        IF VI_Zone_Configs[L_Adaptive_Zone_i].zone >= 1 AND VI_Zone_Configs[L_Adaptive_Zone_i].zone <= 4 THEN
            L_Adaptive_Weight := L_Adaptive_Weight * 1.2;
        ELSIF VI_Zone_Configs[L_Adaptive_Zone_i].zone >= 9 THEN
            L_Adaptive_Weight := L_Adaptive_Weight * 0.7;
        END_IF;

        IF L_Adaptive_Weight > 2.0 THEN
            L_Adaptive_Weight := 2.0;
        ELSIF L_Adaptive_Weight < 0.2 THEN
            L_Adaptive_Weight := 0.2;
        END_IF;

        IF L_Adaptive_Delta > VO_Adaptive_Max_Delta THEN
            VO_Adaptive_Max_Delta := L_Adaptive_Delta;
        END_IF;

        L_Adaptive_Weighted_Sum := L_Adaptive_Weighted_Sum + (L_Adaptive_Delta * L_Adaptive_Weight);
        L_Adaptive_Weight_Total := L_Adaptive_Weight_Total + L_Adaptive_Weight;
    END_IF;
END_FOR;

IF L_Adaptive_Weight_Total > 0.0 THEN
    VO_Adaptive_Effective_Delta := L_Adaptive_Weighted_Sum / L_Adaptive_Weight_Total;
END_IF;

IF VO_Adaptive_Effective_Delta > 1.5 THEN
    VO_Adaptive_Correction := 2.0;
ELSIF VO_Adaptive_Effective_Delta > 0.7 THEN
    VO_Adaptive_Correction := 1.0;
ELSIF VO_Adaptive_Effective_Delta < -1.5 THEN
    VO_Adaptive_Correction := -2.0;
ELSIF VO_Adaptive_Effective_Delta < -0.7 THEN
    VO_Adaptive_Correction := -1.0;
ELSE
    VO_Adaptive_Correction := 0.0;
END_IF;

IF VO_Adaptive_Max_Delta > 2.5 AND VO_Adaptive_Correction < 2.0 THEN
    VO_Adaptive_Correction := 2.0;
END_IF;

VO_Target_Supply_Temp := VO_Target_Supply_Temp + VO_Adaptive_Correction;

IF VO_Target_Supply_Temp < 20.0 THEN
    VO_Target_Supply_Temp := 20.0;
ELSIF VO_Target_Supply_Temp > 45.0 THEN
    VO_Target_Supply_Temp := 45.0;
END_IF;

// >>> BULK_SYNC_ANCHOR: FB_Heating_Adaptive_Target <<<
          
END_FUNCTION_BLOCK

FUNCTION_BLOCK FB_Heating_Circuit_Control
  VAR_INPUT
    VI_System_Time_MS : UDINT;
    VI_Current_Hour : UINT;
    VI_IsActivePLC : BOOL;
    VI_Config : ST_Heating_Config;
    VI_Tariff : ST_Tariff_Config;
    VI_Scenario_Adjust : REAL;
  END_VAR
  VAR_OUTPUT
    VO_Zone_Valves : ARRAY[1..GVL_CONSTANTS.C_MAX_HEATING_CIRCUITS] OF BOOL;
    VO_Heating_Sensor_Fault : BOOL;
  END_VAR
  VAR_IN_OUT
    VI_Zone_Configs : ARRAY[1..GVL_CONSTANTS.C_MAX_HEATING_CIRCUITS] OF ST_FloorHeating_Circuit_Config;
    VI_Floor_Temps : ARRAY[1..GVL_CONSTANTS.C_MAX_HEATING_CIRCUITS] OF REAL;
    VI_Room_Temps : ARRAY[1..16] OF REAL;
    VI_Rule_Actions : ARRAY[1..GVL_CONSTANTS.C_MAX_RULES] OF ST_Rule_Action;
  END_VAR
  VAR
    L_i : INT;
    L_j : INT;
    L_Climate_Zone_ID : INT;
    L_Zone_Config : ST_FloorHeating_Circuit_Config;
    L_Current_Temp : REAL;
    L_Sensor_Error : BOOL;
    L_Floor_Controllers : ARRAY[1..GVL_CONSTANTS.C_MAX_HEATING_CIRCUITS] OF FB_FloorHeating_Controller;
    L_Overheat_Timer : ARRAY[1..GVL_CONSTANTS.C_MAX_HEATING_CIRCUITS] OF FB_System_Timer;
    fbFloorTempValidator : ARRAY[1..GVL_CONSTANTS.C_MAX_HEATING_CIRCUITS] OF FB_Analog_Validator;
    fbRoomTempValidator : ARRAY[1..16] OF FB_Analog_Validator;
  END_VAR

            // ==============================================================================
// Heating circuit control helper
//
// Internal refactoring helper for FB_Heating_System_Manager.
// Owns per-circuit sensor validation, temperature source fallback,
// floor-heating controller call, overheat shutdown, and rule action projection.
// ==============================================================================



VO_Heating_Sensor_Fault := FALSE;

FOR L_i := 1 TO GVL_CONSTANTS.C_MAX_HEATING_CIRCUITS DO
    fbFloorTempValidator[L_i](
        VI_Value := VI_Floor_Temps[L_i],
        VI_Min_Valid := -40.0,
        VI_Max_Valid := 120.0,
        VI_Fallback_Mode := 0
    );

    L_Climate_Zone_ID := VI_Zone_Configs[L_i].zone;
    IF L_Climate_Zone_ID >= 1 AND L_Climate_Zone_ID <= 16 THEN
        fbRoomTempValidator[L_Climate_Zone_ID](
            VI_Value := VI_Room_Temps[L_Climate_Zone_ID],
            VI_Min_Valid := -40.0,
            VI_Max_Valid := 120.0,
            VI_Fallback_Mode := 0
        );
    END_IF;

    // Floor overheat protection
    L_Overheat_Timer[L_i](
        IN := fbFloorTempValidator[L_i].VO_Value > VI_Config.Overheat_Threshold,
        PT := T#60s,
        VI_System_Time_MS := VI_System_Time_MS
    );

    L_Current_Temp := 0.0;
    L_Sensor_Error := FALSE;

    IF VI_Zone_Configs[L_i].control_type = 1 OR VI_Zone_Configs[L_i].control_type = 2 THEN
        // Primary: room air temperature
        IF (L_Climate_Zone_ID >= 1) AND (L_Climate_Zone_ID <= 16) AND (NOT fbRoomTempValidator[L_Climate_Zone_ID].VO_Error) THEN
            L_Current_Temp := fbRoomTempValidator[L_Climate_Zone_ID].VO_Value;
        ELSIF NOT fbFloorTempValidator[L_i].VO_Error THEN
            L_Current_Temp := fbFloorTempValidator[L_i].VO_Value;
        ELSE
            L_Sensor_Error := TRUE;
        END_IF;
    ELSE
        // Primary: floor temperature
        IF NOT fbFloorTempValidator[L_i].VO_Error THEN
            L_Current_Temp := fbFloorTempValidator[L_i].VO_Value;
        ELSIF (L_Climate_Zone_ID >= 1) AND (L_Climate_Zone_ID <= 16) AND (NOT fbRoomTempValidator[L_Climate_Zone_ID].VO_Error) THEN
            L_Current_Temp := fbRoomTempValidator[L_Climate_Zone_ID].VO_Value;
        ELSE
            L_Sensor_Error := TRUE;
        END_IF;
    END_IF;

    IF L_Sensor_Error THEN
        VO_Heating_Sensor_Fault := TRUE;
        VO_Zone_Valves[L_i] := FALSE;
    ELSE
        L_Zone_Config := VI_Zone_Configs[L_i];
        L_Zone_Config.design_temp := L_Zone_Config.design_temp + VI_Scenario_Adjust;

        L_Floor_Controllers[L_i](
            VI_Current_Temp := L_Current_Temp,
            VI_Config := L_Zone_Config,
            VI_Tariff := VI_Tariff,
            VI_Current_Hour := VI_Current_Hour,
            VI_IsActivePLC := VI_IsActivePLC,
            VI_System_Time_MS := VI_System_Time_MS,
            VO_Valve_Bool => VO_Zone_Valves[L_i]
        );
    END_IF;

    IF L_Overheat_Timer[L_i].Q THEN
        VO_Zone_Valves[L_i] := FALSE;
    END_IF;

    FOR L_j := 1 TO GVL_CONSTANTS.C_MAX_RULES DO
        IF VI_Rule_Actions[L_j].Active AND VI_Rule_Actions[L_j].Target_ID = L_i THEN
            IF VI_Rule_Actions[L_j].Action_Type = E_Rule_Action_Type.ACTION_SET_FLOOR_HEATING THEN
                VO_Zone_Valves[L_i] := (VI_Rule_Actions[L_j].Value > 0.5);
            END_IF;
        END_IF;
    END_FOR;
END_FOR;

// >>> BULK_SYNC_ANCHOR: FB_Heating_Circuit_Control <<<
          
END_FUNCTION_BLOCK

FUNCTION_BLOCK FB_Rule_Engine
  VAR_INPUT
    VI_System_Time_MS : UDINT;
    VI_IsActivePLC : BOOL;
    VI_Security_Armed : BOOL;
    VI_Current_Time : TOD;
    VI_Day_Of_Week : INT;
  END_VAR
  VAR_OUTPUT
    VO_Preheat_Request : BOOL;
    VO_Actions : ARRAY[1..GVL_CONSTANTS.C_MAX_RULES] OF ST_Rule_Action;
  END_VAR
  VAR_IN_OUT
    VI_Rules : ARRAY[1..GVL_CONSTANTS.C_MAX_RULES] OF ST_User_Rule;
    VI_Indoor_Temps : ARRAY[1..16] OF REAL;
    VI_Floor_Temps : ARRAY[1..8] OF REAL;
    VI_Humidities : ARRAY[1..16] OF REAL;
    VI_CO2_Levels : ARRAY[1..16] OF REAL;
    VI_Motion_Sensors : ARRAY[1..16] OF BOOL;
    VI_Door_Sensors : ARRAY[1..GVL_CONSTANTS.C_MAX_DOOR_SENSORS] OF BOOL;
    VI_Window_Sensors : ARRAY[1..16] OF BOOL;
    VI_Water_Sensors : ARRAY[1..GVL_CONSTANTS.C_MAX_FLOOD_SENSORS] OF BOOL;
    VI_Smoke_Sensors : ARRAY[1..GVL_CONSTANTS.C_MAX_SMOKE_SENSORS] OF BOOL;
    VI_Methane_Sensors : ARRAY[1..GVL_CONSTANTS.C_MAX_METHANE_SENSORS] OF REAL;
    VI_CO_Sensors : ARRAY[1..GVL_CONSTANTS.C_MAX_CO_SENSORS] OF REAL;
  END_VAR
  VAR
    L_i : INT;
    L_Condition_Met : BOOL;
    L_Current_Value : REAL;
    L_Triggers : ARRAY[1..GVL_CONSTANTS.C_MAX_RULES] OF R_TRIG;
    L_Trigger_Count : ARRAY[1..GVL_CONSTANTS.C_MAX_RULES] OF UINT;
    L_Last_Reset_Time : UDINT;
    L_Elapsed_Time : UDINT;
  END_VAR

            IF NOT VI_IsActivePLC THEN RETURN; END_IF;

VO_Preheat_Request := FALSE;


// Сброс счетчиков срабатываний каждую минуту (защита от циклических зависимостей/дребезга)
L_Elapsed_Time := (SEL(VI_System_Time_MS >= L_Last_Reset_Time, VI_System_Time_MS - L_Last_Reset_Time, (4294967295 - L_Last_Reset_Time) + VI_System_Time_MS + 1));

IF L_Elapsed_Time >= GVL_CONSTANTS.C_MS_IN_MINUTE THEN
    L_Last_Reset_Time := VI_System_Time_MS;
    FOR L_i := 1 TO GVL_CONSTANTS.C_MAX_RULES DO
        L_Trigger_Count[L_i] := 0;
    END_FOR;
END_IF;

FOR L_i := 1 TO GVL_CONSTANTS.C_MAX_RULES DO

    VO_Actions[L_i].Active := FALSE;
    IF VI_Rules[L_i].Enabled THEN
        L_Condition_Met := FALSE;
        L_Current_Value := 0.0;
        
        // Определение значения для проверки
        IF VI_Rules[L_i].Condition_Target_ID > 0 THEN
            CASE VI_Rules[L_i].Condition_Type OF
                E_Rule_Condition_Type.COND_AIR_TEMP: IF VI_Rules[L_i].Condition_Target_ID <= 16 THEN L_Current_Value := VI_Indoor_Temps[VI_Rules[L_i].Condition_Target_ID]; END_IF;
                E_Rule_Condition_Type.COND_FLOOR_TEMP: IF VI_Rules[L_i].Condition_Target_ID <= 8 THEN L_Current_Value := VI_Floor_Temps[VI_Rules[L_i].Condition_Target_ID]; END_IF;
                E_Rule_Condition_Type.COND_HUMIDITY: IF VI_Rules[L_i].Condition_Target_ID <= 16 THEN L_Current_Value := VI_Humidities[VI_Rules[L_i].Condition_Target_ID]; END_IF;
                E_Rule_Condition_Type.COND_CO2: IF VI_Rules[L_i].Condition_Target_ID <= 16 THEN L_Current_Value := VI_CO2_Levels[VI_Rules[L_i].Condition_Target_ID]; END_IF;
                E_Rule_Condition_Type.COND_MOTION: IF VI_Rules[L_i].Condition_Target_ID <= 16 THEN L_Current_Value := SEL(VI_Motion_Sensors[VI_Rules[L_i].Condition_Target_ID], 0.0, 1.0); END_IF;
                E_Rule_Condition_Type.COND_DOOR_WINDOW: 
                    IF VI_Rules[L_i].Condition_Target_ID <= GVL_CONSTANTS.C_MAX_DOOR_SENSORS THEN
                        L_Current_Value := SEL(VI_Door_Sensors[VI_Rules[L_i].Condition_Target_ID] OR VI_Window_Sensors[VI_Rules[L_i].Condition_Target_ID], 0.0, 1.0);
                    ELSIF VI_Rules[L_i].Condition_Target_ID <= 16 THEN
                        L_Current_Value := SEL(VI_Window_Sensors[VI_Rules[L_i].Condition_Target_ID], 0.0, 1.0);
                    END_IF;
                E_Rule_Condition_Type.COND_FLOOD: IF VI_Rules[L_i].Condition_Target_ID <= GVL_CONSTANTS.C_MAX_FLOOD_SENSORS THEN L_Current_Value := SEL(VI_Water_Sensors[VI_Rules[L_i].Condition_Target_ID], 0.0, 1.0); END_IF;
                E_Rule_Condition_Type.COND_SMOKE: IF VI_Rules[L_i].Condition_Target_ID <= GVL_CONSTANTS.C_MAX_SMOKE_SENSORS THEN L_Current_Value := SEL(VI_Smoke_Sensors[VI_Rules[L_i].Condition_Target_ID], 0.0, 1.0); END_IF;
                E_Rule_Condition_Type.COND_METHANE: IF VI_Rules[L_i].Condition_Target_ID <= GVL_CONSTANTS.C_MAX_METHANE_SENSORS THEN L_Current_Value := VI_Methane_Sensors[VI_Rules[L_i].Condition_Target_ID]; END_IF;
                E_Rule_Condition_Type.COND_CO: IF VI_Rules[L_i].Condition_Target_ID <= GVL_CONSTANTS.C_MAX_CO_SENSORS THEN L_Current_Value := VI_CO_Sensors[VI_Rules[L_i].Condition_Target_ID]; END_IF;
                E_Rule_Condition_Type.COND_TIME_OF_DAY: L_Current_Value := TO_REAL(TOD_TO_UDINT(VI_Current_Time) / GVL_CONSTANTS.C_MS_IN_MINUTE); // Время в минутах
                E_Rule_Condition_Type.COND_DAY_OF_WEEK: L_Current_Value := TO_REAL(VI_Day_Of_Week);
            END_CASE;
        ELSE
            IF VI_Rules[L_i].Condition_Type = E_Rule_Condition_Type.COND_TIME_OF_DAY THEN
                L_Current_Value := TO_REAL(TOD_TO_UDINT(VI_Current_Time) / GVL_CONSTANTS.C_MS_IN_MINUTE); // Время в минутах
            ELSIF VI_Rules[L_i].Condition_Type = E_Rule_Condition_Type.COND_DAY_OF_WEEK THEN
                L_Current_Value := TO_REAL(VI_Day_Of_Week);
            END_IF;
        END_IF;
        
        // Проверка условия
        CASE VI_Rules[L_i].Condition_Op OF
            E_Rule_Comparison.COMP_GT: L_Condition_Met := (L_Current_Value > VI_Rules[L_i].Condition_Value);
            E_Rule_Comparison.COMP_LT: L_Condition_Met := (L_Current_Value < VI_Rules[L_i].Condition_Value);
            E_Rule_Comparison.COMP_EQ: L_Condition_Met := (ABS(L_Current_Value - VI_Rules[L_i].Condition_Value) < 0.1);
            E_Rule_Comparison.COMP_GE: L_Condition_Met := (L_Current_Value >= VI_Rules[L_i].Condition_Value);
            E_Rule_Comparison.COMP_LE: L_Condition_Met := (L_Current_Value <= VI_Rules[L_i].Condition_Value);
            E_Rule_Comparison.COMP_IN_RANGE: L_Condition_Met := (L_Current_Value >= VI_Rules[L_i].Condition_Value) AND (L_Current_Value <= VI_Rules[L_i].Condition_Value_Max);
            E_Rule_Comparison.COMP_TRUE: L_Condition_Met := (L_Current_Value > 0.5);
            E_Rule_Comparison.COMP_FALSE: L_Condition_Met := (L_Current_Value < 0.5);
        END_CASE;
        
        // Формирование действия
        L_Triggers[L_i](CLK := L_Condition_Met);
        
        IF L_Triggers[L_i].Q THEN
            L_Trigger_Count[L_i] := L_Trigger_Count[L_i] + 1;
            IF L_Trigger_Count[L_i] > 10 THEN
                // ТЗ 13.5: Блокировка правила при слишком частом срабатывании (циклическая зависимость)
                VO_Actions[L_i].Active := FALSE;
                VO_Actions[L_i].Triggered := FALSE;
                CONTINUE; // Пропускаем выполнение
            END_IF;
        END_IF;
        
        IF L_Condition_Met AND (L_Trigger_Count[L_i] <= 10) THEN
            VO_Actions[L_i].Active := TRUE;
            VO_Actions[L_i].Triggered := L_Triggers[L_i].Q;
            VO_Actions[L_i].Action_Type := VI_Rules[L_i].Action_Type;
            VO_Actions[L_i].Target_ID := VI_Rules[L_i].Action_Target_ID;
            VO_Actions[L_i].Value := VI_Rules[L_i].Action_Value;
        END_IF;
    END_IF;
END_FOR;
// >>> BULK_SYNC_ANCHOR: FB_Rule_Engine <<<
          
END_FUNCTION_BLOCK

FUNCTION_BLOCK FB_Trend_Analyzer
  VAR_INPUT
    VI_Count : INT;
  END_VAR
  VAR_OUTPUT
    VO_Average : REAL;
    VO_Max : REAL;
    VO_Min : REAL;
    VO_Trend_Up : BOOL;
    VO_Trend_Down : BOOL;
  END_VAR
  VAR_IN_OUT
    VI_Data : ARRAY[1..GVL_CONSTANTS.C_MAX_TREND_DATA_POINTS] OF REAL;
  END_VAR
  VAR
    L_i : INT;
    L_Sum : REAL;
  END_VAR

            IF VI_Count > 0 AND VI_Count <= GVL_CONSTANTS.C_MAX_TREND_DATA_POINTS THEN
    VO_Max := VI_Data[1];
    VO_Min := VI_Data[1];
    L_Sum := 0.0;
    
    FOR L_i := 1 TO VI_Count DO
        IF VI_Data[L_i] > VO_Max THEN VO_Max := VI_Data[L_i]; END_IF;
        IF VI_Data[L_i] < VO_Min THEN VO_Min := VI_Data[L_i]; END_IF;
        L_Sum := L_Sum + VI_Data[L_i];
    END_FOR;
    
    VO_Average := L_Sum / INT_TO_REAL(VI_Count);
    
    IF VI_Count >= 2 THEN
        VO_Trend_Up := (VI_Data[VI_Count] > VI_Data[1]);
        VO_Trend_Down := (VI_Data[VI_Count] < VI_Data[1]);
    END_IF;
END_IF;
          
END_FUNCTION_BLOCK

FUNCTION_BLOCK FB_BlackBox_Recorder
  VAR_INPUT
    VI_Current_Data : ST_BlackBox_Record;
    VI_Freeze : BOOL;
  END_VAR
  VAR_OUTPUT
    VO_Frozen : BOOL;
    VO_Records_Count : INT;
  END_VAR
  VAR
    L_Write_Index : INT := 0;
    L_Initialized : BOOL := FALSE;
  END_VAR

            IF NOT L_Initialized THEN
    L_Write_Index := GVL_Retain.G_BlackBox_LastIndex;
    IF L_Write_Index < 0 OR L_Write_Index >= GVL_CONSTANTS.C_MAX_BLACKBOX_RECORDS THEN
        L_Write_Index := 0;
        GVL_Retain.G_BlackBox_LastIndex := 0;
    END_IF;
    L_Initialized := TRUE;
END_IF;

IF VI_Freeze THEN
    GVL_Retain.G_BlackBox_Frozen := TRUE;
END_IF;

VO_Frozen := GVL_Retain.G_BlackBox_Frozen;

IF NOT GVL_Retain.G_BlackBox_Frozen THEN
    GVL_Retain.G_BlackBox_Buffer[L_Write_Index] := VI_Current_Data;
    GVL_Retain.G_BlackBox_LastIndex := L_Write_Index;
    
    L_Write_Index := L_Write_Index + 1;
    IF L_Write_Index >= GVL_CONSTANTS.C_MAX_BLACKBOX_RECORDS THEN
        L_Write_Index := 0;
    END_IF;
END_IF;

VO_Records_Count := GVL_CONSTANTS.C_MAX_BLACKBOX_RECORDS; // Размер кольцевого буфера
// >>> BULK_SYNC_ANCHOR: FB_BlackBox_Recorder <<<
          
END_FUNCTION_BLOCK

FUNCTION_BLOCK FB_System_Init
  VAR_IN_OUT
    VIO_Local_State : ST_System_State_Snapshot;
    VIO_Remote_State : ST_System_State_Snapshot;
  END_VAR
  VAR
    L_i : INT;
  END_VAR

            // ==============================================================================
// System init helper
//
// Internal helper for PRG_System.
// Owns first-boot initialization of RETAIN runtime state.
// ==============================================================================



IF NOT GVL_Retain.G_Initialized THEN
    FOR L_i := 0 TO GVL_CONSTANTS.C_MAX_PRESENCE_HISTORY - 1 DO
        GVL_Retain.G_Presence_History[L_i] := 0;
    END_FOR;

    GVL_Retain.G_History_Write_Idx := 1;
    GVL_Retain.G_History_Total_Events := 0;

    FOR L_i := 1 TO GVL_CONSTANTS.C_MAX_BOILERS DO
        GVL_Retain.G_Boiler_Accumulated_MS[L_i] := 0;
        GVL_Retain.G_Boiler_Work_Seconds[L_i] := 0;
    END_FOR;

    FOR L_i := 1 TO GVL_CONSTANTS.C_MAX_MANIFOLDS DO
        GVL_Retain.G_Valve_Test_Results[L_i] := FALSE;
    END_FOR;

    VIO_Local_State.Version := 0;
    VIO_Remote_State.Version := 0;

    GVL_Retain.G_Initialized := TRUE;
END_IF;

// >>> BULK_SYNC_ANCHOR: FB_System_Init <<<
          
END_FUNCTION_BLOCK

FUNCTION_BLOCK FB_Safety_Manager
  VAR_INPUT
    VI_Gas_Alarm : BOOL;
    VI_Leak_Alarm : BOOL;
    VI_Smoke_Alarm : BOOL;
    VI_Reset : BOOL;
  END_VAR
  VAR_OUTPUT
    VO_Gas_Latched : BOOL;
    VO_Leak_Latched : BOOL;
    VO_Smoke_Latched : BOOL;
    VO_Emergency_Stop : BOOL;
  END_VAR
  VAR
    L_Any_Active : BOOL;
  END_VAR

            // Защёлкиваем аварии независимо друг от друга
IF VI_Gas_Alarm THEN
    VO_Gas_Latched := TRUE;
END_IF;

IF VI_Leak_Alarm THEN
    VO_Leak_Latched := TRUE;
END_IF;

IF VI_Smoke_Alarm THEN
    VO_Smoke_Latched := TRUE;
END_IF;

L_Any_Active := VI_Gas_Alarm OR VI_Leak_Alarm OR VI_Smoke_Alarm;

// Ручной сброс допустим только когда все входные аварийные сигналы уже исчезли
IF VI_Reset AND NOT L_Any_Active THEN
    VO_Gas_Latched := FALSE;
    VO_Leak_Latched := FALSE;
    VO_Smoke_Latched := FALSE;
END_IF;

// Агрегированный аварийный стоп = любая защёлкнутая safety-авария
VO_Emergency_Stop := VO_Gas_Latched OR VO_Leak_Latched OR VO_Smoke_Latched;

// >>> BULK_SYNC_ANCHOR: FB_Safety_Manager <<<
          
END_FUNCTION_BLOCK

FUNCTION_BLOCK FB_System_Recovery
  VAR_IN_OUT
    VIO_Recovery_Done : BOOL;
  END_VAR

            // ==============================================================================
// System recovery helper
//
// Internal helper for PRG_System.
// Owns one-shot recovery of persistent safety/system state after boot.
// ==============================================================================



IF NOT VIO_Recovery_Done THEN
    IF GVL_PERSISTENT.P_Valid THEN
        GVL_STATE.G_Safety_Gas_Latched := GVL_PERSISTENT.P_Safety_Gas_Latched;
        GVL_STATE.G_Safety_Smoke_Latched := GVL_PERSISTENT.P_Safety_Smoke_Latched;
        GVL_STATE.G_Safety_Leak_Latched := GVL_PERSISTENT.P_Safety_Leak_Latched;
        GVL_STATE.G_System_Mode := GVL_PERSISTENT.P_System_Mode;
    END_IF;

    VIO_Recovery_Done := TRUE;
END_IF;

// >>> BULK_SYNC_ANCHOR: FB_System_Recovery <<<
          
END_FUNCTION_BLOCK

FUNCTION_BLOCK FB_System_Coordinator
  VAR_INPUT
    VI_Fire_Latched : BOOL;
    VI_Gas_Latched : BOOL;
    VI_Leak_Latched : BOOL;
    VI_IO_Degraded : BOOL;
    VI_Ownership_Violation : BOOL;
    VI_Behavior_Mode : E_Behavior_Mode;
  END_VAR
  VAR_OUTPUT
    VO_Block_Heating : BOOL;
    VO_Block_Ventilation : BOOL;
    VO_Block_Lighting : BOOL;
    VO_Block_Sockets : BOOL;
    VO_System_Degraded : BOOL;
    VO_Code : UDINT;
  END_VAR

            // reset
VO_Block_Heating := FALSE;
VO_Block_Ventilation := FALSE;
VO_Block_Lighting := FALSE;
VO_Block_Sockets := FALSE;
VO_System_Degraded := FALSE;
VO_Code := 0;

// FIRE has highest priority. Safety-stop ownership remains in PRG_Safety.
IF VI_Fire_Latched THEN
    VO_Block_Heating := TRUE;
    VO_Block_Ventilation := TRUE;
    VO_Block_Sockets := TRUE;
    VO_Code := 100;
    RETURN;
END_IF;

// GAS has higher priority than behavior mode.
IF VI_Gas_Latched THEN
    VO_Block_Heating := TRUE;
    VO_Block_Lighting := TRUE;
    VO_Block_Sockets := TRUE;
    VO_Code := 200;
    RETURN;
END_IF;

// LEAK blocks heating but does not suppress later degradation/mode overlays.
IF VI_Leak_Latched THEN
    VO_Block_Heating := TRUE;
    VO_Code := 300;
END_IF;

// IO degraded blocks heating and marks system degraded.
IF VI_IO_Degraded THEN
    VO_System_Degraded := TRUE;
    VO_Block_Heating := TRUE;
    IF VO_Code = 0 THEN
        VO_Code := 400;
    END_IF;
END_IF;

// Ownership violation marks system degraded. Test/result handler owns any safe-stop reaction.
IF VI_Ownership_Violation THEN
    VO_System_Degraded := TRUE;
    IF VO_Code = 0 THEN
        VO_Code := 500;
    END_IF;
END_IF;

// Behavior mode overlays. These are lower priority than safety/system faults.
CASE VI_Behavior_Mode OF
    BEHAVIOR_AWAY:
        VO_Block_Lighting := TRUE;
        VO_Block_Sockets := TRUE;
        IF VO_Code = 0 THEN
            VO_Code := 600;
        END_IF;

    BEHAVIOR_NIGHT:
        VO_Block_Lighting := TRUE;
        IF VO_Code = 0 THEN
            VO_Code := 700;
        END_IF;

    BEHAVIOR_MAINTENANCE:
        VO_Block_Heating := TRUE;
        VO_Block_Ventilation := TRUE;
        IF VO_Code = 0 THEN
            VO_Code := 800;
        END_IF;
END_CASE;
          
END_FUNCTION_BLOCK

FUNCTION_BLOCK FB_System_Diagnostics

            // ==============================================================================
// System diagnostics helper
//
// Internal helper for PRG_System.
// Owns diagnostic flag export into GVL_STATUS.G_Diagnostics.
// ==============================================================================


GVL_STATUS.G_Diagnostics.Sensor_Fault :=
    GVL_STATE.G_Heating_Sensor_Fault OR
    GVL_STATE.G_DHW_Sensor_Fault OR
    GVL_STATUS.G_Diagnostics.Manifold_Pressure_Fault_Active OR
    GVL_STATUS.G_Diagnostics.Manifold_Current_Fault_Active OR
    GVL_STATUS.G_Diagnostics.Manifold_Return_Temp_Fault_Active;

GVL_STATUS.G_Diagnostics.IO_Offline :=
    GVL_STATE.G_Heating_IO_Fault OR
    GVL_STATE.G_DHW_IO_Fault OR
    GVL_STATE.G_Ventilation_IO_Fault OR
    GVL_STATE.G_Lighting_IO_Fault;

GVL_STATUS.G_Diagnostics.Subsystem_Degraded :=
    GVL_STATE.G_Heating_Subsystem_Degraded OR
    GVL_STATE.G_DHW_Subsystem_Degraded OR
    GVL_STATE.G_Ventilation_Subsystem_Degraded OR
    GVL_STATUS.G_Diagnostics.Manifold_Pressure_Fault_Active OR
    GVL_STATUS.G_Diagnostics.Manifold_Current_Fault_Active OR
    GVL_STATUS.G_Diagnostics.Manifold_Return_Temp_Fault_Active;

// >>> BULK_SYNC_ANCHOR: FB_System_Diagnostics <<<
          
END_FUNCTION_BLOCK

FUNCTION_BLOCK FB_Heating_System_Manager
  VAR_INPUT
    VI_Preheat_Request : BOOL;
    L_Climate_Zone_ID : INT;
    VI_System_Mode : E_System_Operating_Mode;
    VI_System_Time_MS : UDINT;
    VI_Current_TOD : TOD;
    VI_IsActivePLC : BOOL;
    VI_Outdoor_Temp : REAL;
    VI_Config : ST_Heating_Config;
    VI_Tariff : ST_Tariff_Config;
    VI_Current_Hour : UINT;
    VI_Boiler_Stop : BOOL;
    VI_DHW_Heating_Demand : BOOL;
    VI_DHW_Target_Temp : REAL;
    VI_Current_Scenario : E_SCENARIO_TYPE;
    VI_Emergency_Stop : BOOL;
    VI_Gas_Safety_Stop : BOOL;
    VI_Boiler_Error_Status : ARRAY[1..GVL_CONSTANTS.C_MAX_BOILERS] OF BOOL;
    VI_Boiler_OT_Online : ARRAY[1..GVL_CONSTANTS.C_MAX_BOILERS] OF BOOL;
    VI_Boiler_Modulation : ARRAY[1..GVL_CONSTANTS.C_MAX_BOILERS] OF REAL;
  END_VAR
  VAR_OUTPUT
    VO_Manifold_Valves : ARRAY[1..GVL_CONSTANTS.C_MAX_MANIFOLDS] OF REAL;
    VO_Manifold_Pumps : ARRAY[1..GVL_CONSTANTS.C_MAX_MANIFOLDS] OF BOOL;
    VO_Zone_Valves : ARRAY[1..GVL_CONSTANTS.C_MAX_HEATING_CIRCUITS] OF BOOL;
    VO_Boiler_OT_Enable : ARRAY[1..GVL_CONSTANTS.C_MAX_BOILERS] OF BOOL;
    VO_Boiler_OT_Setpoint : ARRAY[1..GVL_CONSTANTS.C_MAX_BOILERS] OF REAL;
    VO_Backup_Circulation_Pump : BOOL;
    VO_Electric_Heater_Enable : BOOL;
    VO_Freeze_Risk_Status : BOOL;
    VO_Status : ARRAY[1..GVL_CONSTANTS.C_MAX_MANIFOLDS] OF ST_Manifold_Status;
    VO_Boiler_Status : ARRAY[1..GVL_CONSTANTS.C_MAX_BOILERS] OF ST_Boiler_Status;
  END_VAR
  VAR_IN_OUT
    VI_Floor_Temps : ARRAY[1..GVL_CONSTANTS.C_MAX_HEATING_CIRCUITS] OF REAL;
    VI_Room_Temps : ARRAY[1..16] OF REAL;
    VI_Manifold_Pressures : ARRAY[1..GVL_CONSTANTS.C_MAX_MANIFOLDS] OF REAL;
    VI_Manifold_Currents : ARRAY[1..GVL_CONSTANTS.C_MAX_MANIFOLDS] OF REAL;
    VI_Manifold_Temps_Supply : ARRAY[1..GVL_CONSTANTS.C_MAX_MANIFOLDS] OF REAL;
    VI_Manifold_Temps_Return : ARRAY[1..GVL_CONSTANTS.C_MAX_MANIFOLDS] OF REAL;
    VI_Boiler_Flame_Status : ARRAY[1..GVL_CONSTANTS.C_MAX_BOILERS] OF BOOL;
    VI_Zone_Configs : ARRAY[1..GVL_CONSTANTS.C_MAX_HEATING_CIRCUITS] OF ST_FloorHeating_Circuit_Config;
    VI_Rule_Actions : ARRAY[1..GVL_CONSTANTS.C_MAX_RULES] OF ST_Rule_Action;
    VI_IO_Modules_Online : ARRAY[1..GVL_CONSTANTS.C_MAX_MODULES] OF BOOL;
    VI_Scenario_Configs : ARRAY[1..GVL_CONSTANTS.C_MAX_SCENARIOS] OF ST_Scenario_Config;
    VI_Manifold_End_Switches : ARRAY[1..GVL_CONSTANTS.C_MAX_MANIFOLDS] OF BOOL;
    VI_Valve_Test_Config : ARRAY[1..GVL_CONSTANTS.C_MAX_MANIFOLDS] OF ST_Valve_Test_Config;
  END_VAR
  VAR
    L_Lead_Boiler : BYTE := 1;
    L_i : INT;
    L_j : INT;
    L_Target_Supply_Temp : REAL;
    L_Demand_Power : REAL;
    L_Any_Zone_Active : ARRAY[1..GVL_CONSTANTS.C_MAX_MANIFOLDS] OF BOOL;
    L_Prev_Scenario : E_SCENARIO_TYPE;
    L_Scenario_Adjust : REAL;
    L_Target_Scenario_Adjust : REAL;
    L_Transition_Temp : FB_Scenario_Transition_Controller;
    fbValveTestManager : FB_Valve_Test_Manager;
    L_IO_Failsafe_Active : BOOL;
    L_Freeze_Mode_Active : BOOL;
    L_Freeze_Target_Supply : REAL;
    L_Min_Supply_Temp : REAL;
    L_Policy_Degraded : BOOL;
    L_Any_Sensor_Error : BOOL;
    L_Any_Subsystem_Degraded : BOOL;
    L_Adaptive_Max_Delta : REAL;
    L_Adaptive_Effective_Delta : REAL;
    L_Adaptive_Correction : REAL;
    fbAdaptiveTarget : FB_Heating_Adaptive_Target;
    fbSafetyGate : FB_Heating_Safety_Gate;
    fbCircuitControl : FB_Heating_Circuit_Control;
    fbManifoldControl : FB_Heating_Manifold_Control;
    fbBoilerControl : FB_Heating_Boiler_Control;
  END_VAR

            // ==============================================================================
// Блок управления системой отопления (Heating System Manager)
// Назначение:
// - Публичный фасад системы отопления.
// - Оркестрация доменных FB отопления.
// - Проекция безопасных состояний на физические выходы.
// - Интеграция с Rule Engine, HMI status и GVL_STATE.
// ==============================================================================



// ========================================
// Policy and fault pre-scan
// ========================================
L_Policy_Degraded := (VI_System_Mode = E_System_Operating_Mode.MODE_DEGRADED);

GVL_STATE.G_Heating_IO_Fault := FALSE;
GVL_STATE.G_Heating_Sensor_Fault := FALSE;
GVL_STATE.G_Heating_Subsystem_Degraded := FALSE;
L_Any_Sensor_Error := FALSE;
L_Any_Subsystem_Degraded := FALSE;

L_IO_Failsafe_Active := FALSE;
FOR L_i := 1 TO GVL_CONSTANTS.C_MAX_MODULES DO
    IF NOT VI_IO_Modules_Online[L_i] THEN
        L_IO_Failsafe_Active := TRUE;
        GVL_STATE.G_Heating_IO_Fault := TRUE;
        GVL_STATE.G_Heating_Subsystem_Degraded := TRUE;
        EXIT;
    END_IF;
END_FOR;

fbSafetyGate(
    VI_System_Mode := VI_System_Mode,
    VI_Emergency_Stop := VI_Emergency_Stop,
    VI_Gas_Safety_Stop := VI_Gas_Safety_Stop,
    VI_IO_Failsafe_Active := L_IO_Failsafe_Active,
    VI_Outdoor_Temp := VI_Outdoor_Temp,
    VI_Freeze_Threshold := VI_Config.Freeze_Threshold,
    VI_Floor_Temps := VI_Floor_Temps,
    VO_Freeze_Mode_Active => L_Freeze_Mode_Active,
    VO_Freeze_Target_Supply => L_Freeze_Target_Supply
);

// ========================================
// Safe-state output projection
// ========================================
VO_Backup_Circulation_Pump := FALSE;
VO_Electric_Heater_Enable := FALSE;
VO_Freeze_Risk_Status := FALSE;

IF fbSafetyGate.VO_Block_Normal_Heating THEN
    FOR L_i := 1 TO GVL_CONSTANTS.C_MAX_HEATING_CIRCUITS DO
        VO_Zone_Valves[L_i] := FALSE;
    END_FOR;

    FOR L_i := 1 TO GVL_CONSTANTS.C_MAX_MANIFOLDS DO
        IF fbSafetyGate.VO_IO_Failsafe_Active AND L_Freeze_Mode_Active THEN
            VO_Manifold_Pumps[L_i] := TRUE;
            VO_Manifold_Valves[L_i] := 35.0;
        ELSE
            VO_Manifold_Pumps[L_i] := FALSE;
            VO_Manifold_Valves[L_i] := 0.0;
        END_IF;
    END_FOR;

    FOR L_i := 1 TO GVL_CONSTANTS.C_MAX_BOILERS DO
        VO_Boiler_OT_Enable[L_i] := FALSE;
        VO_Boiler_OT_Setpoint[L_i] := 0.0;
        VO_Boiler_Status[L_i].Warning := FALSE;
        VO_Boiler_Status[L_i].Error := TRUE;
    END_FOR;

    IF fbSafetyGate.VO_Gas_Safety_Active AND L_Freeze_Mode_Active THEN
        VO_Backup_Circulation_Pump := TRUE;
        L_Min_Supply_Temp := 1000.0;
        FOR L_i := 1 TO GVL_CONSTANTS.C_MAX_MANIFOLDS DO
            IF VI_Manifold_Temps_Supply[L_i] < L_Min_Supply_Temp THEN
                L_Min_Supply_Temp := VI_Manifold_Temps_Supply[L_i];
            END_IF;
        END_FOR;
        IF L_Min_Supply_Temp > 900.0 THEN
            L_Min_Supply_Temp := 0.0;
        END_IF;

        IF L_Min_Supply_Temp < (L_Freeze_Target_Supply - 1.0) THEN
            VO_Electric_Heater_Enable := TRUE;
        ELSIF L_Min_Supply_Temp > (L_Freeze_Target_Supply + 1.0) THEN
            VO_Electric_Heater_Enable := FALSE;
        END_IF;

        // При защёлкнутой газовой аварии оператор должен видеть, что система живёт в деградированном anti-freeze режиме.
        VO_Freeze_Risk_Status := TRUE;
    END_IF;

    IF fbSafetyGate.VO_IO_Failsafe_Active AND L_Freeze_Mode_Active THEN
        IF VI_Boiler_OT_Online[1] AND NOT VI_Boiler_Error_Status[1] THEN
            VO_Boiler_OT_Enable[1] := TRUE;
            VO_Boiler_OT_Setpoint[1] := L_Freeze_Target_Supply;
        END_IF;
    END_IF;

    RETURN;
END_IF;

// --- ADAPTIVE TARGET ---
fbAdaptiveTarget(
    VI_Base_Target_Supply_Temp := L_Target_Supply_Temp,
    VI_Global_Target_Temperature := GVL_STATE.G_Target_Temperature,
    VI_Zone_Configs := VI_Zone_Configs,
    VI_Floor_Temps := VI_Floor_Temps,
    VI_Room_Temps := VI_Room_Temps,
    VO_Target_Supply_Temp => L_Target_Supply_Temp,
    VO_Adaptive_Correction => L_Adaptive_Correction,
    VO_Adaptive_Effective_Delta => L_Adaptive_Effective_Delta,
    VO_Adaptive_Max_Delta => L_Adaptive_Max_Delta
);

// --- CIRCUIT CONTROL ---
fbCircuitControl(
    VI_System_Time_MS := VI_System_Time_MS,
    VI_Current_Hour := VI_Current_Hour,
    VI_IsActivePLC := VI_IsActivePLC,
    VI_Config := VI_Config,
    VI_Tariff := VI_Tariff,
    VI_Scenario_Adjust := L_Scenario_Adjust,
    VI_Zone_Configs := VI_Zone_Configs,
    VI_Floor_Temps := VI_Floor_Temps,
    VI_Room_Temps := VI_Room_Temps,
    VI_Rule_Actions := VI_Rule_Actions,
    VO_Zone_Valves => VO_Zone_Valves,
    VO_Heating_Sensor_Fault => L_Any_Sensor_Error
);

GVL_STATE.G_Heating_Sensor_Fault := L_Any_Sensor_Error;

// --- MANIFOLD DEMAND MAP ---
FOR L_i := 1 TO GVL_CONSTANTS.C_MAX_MANIFOLDS DO
    L_Any_Zone_Active[L_i] := FALSE;
END_FOR;

FOR L_i := 1 TO GVL_CONSTANTS.C_MAX_HEATING_CIRCUITS DO
    IF VO_Zone_Valves[L_i] THEN
        L_j := VI_Zone_Configs[L_i].manifold_id;
        IF L_j >= 1 AND L_j <= GVL_CONSTANTS.C_MAX_MANIFOLDS THEN
            L_Any_Zone_Active[L_j] := TRUE;
        END_IF;
    END_IF;
END_FOR;

// --- MANIFOLD CONTROL ---
fbManifoldControl(
    VI_System_Time_MS := VI_System_Time_MS,
    VI_IsActivePLC := VI_IsActivePLC,
    VI_DHW_Heating_Demand := VI_DHW_Heating_Demand,
    VI_Freeze_Mode_Active := L_Freeze_Mode_Active,
    VI_Target_Supply_Temp := L_Target_Supply_Temp,
    VI_Any_Zone_Active := L_Any_Zone_Active,
    VI_Manifold_Pressures := VI_Manifold_Pressures,
    VI_Manifold_Currents := VI_Manifold_Currents,
    VI_Manifold_Temps_Supply := VI_Manifold_Temps_Supply,
    VI_Manifold_Temps_Return := VI_Manifold_Temps_Return,
    VO_Manifold_Pumps => VO_Manifold_Pumps,
    VO_Manifold_Valves => VO_Manifold_Valves,
    VO_Status => VO_Status
);

// --- VALVE TEST OVERRIDE ---
fbValveTestManager(
    VI_System_Time_MS := VI_System_Time_MS,
    VI_IsActivePLC := VI_IsActivePLC,
    VI_Valve_Currents := VI_Manifold_Currents,
    VI_Valve_End_Switches := VI_Manifold_End_Switches,
    VI_Config := VI_Valve_Test_Config
);

IF fbValveTestManager.VO_Test_Active THEN
    L_i := fbValveTestManager.VO_Current_Valve;
    IF L_i >= 1 AND L_i <= GVL_CONSTANTS.C_MAX_MANIFOLDS THEN
        IF fbValveTestManager.VO_Valve_Cmd[L_i] THEN
            VO_Manifold_Valves[L_i] := 100.0;
        ELSE
            VO_Manifold_Valves[L_i] := 0.0;
        END_IF;
        VO_Manifold_Pumps[L_i] := FALSE; // Отключаем насос при тестировании клапана
    END_IF;
END_IF;

// --- BOILER CONTROL ---
fbBoilerControl(
    VI_System_Time_MS := VI_System_Time_MS,
    VI_IsActivePLC := VI_IsActivePLC,
    VI_DHW_Heating_Demand := VI_DHW_Heating_Demand,
    VI_DHW_Target_Temp := VI_DHW_Target_Temp,
    VI_Target_Supply_Temp := L_Target_Supply_Temp,
    VI_Freeze_Mode_Active := L_Freeze_Mode_Active,
    VI_Policy_Degraded := L_Policy_Degraded,
    VI_Manifold_Pumps := VO_Manifold_Pumps,
    VI_Manifold_Valves := VO_Manifold_Valves,
    VI_Boiler_Flame_Status := VI_Boiler_Flame_Status,
    VI_Boiler_Error_Status := VI_Boiler_Error_Status,
    VI_Boiler_OT_Online := VI_Boiler_OT_Online,
    VI_Boiler_Modulation := VI_Boiler_Modulation,
    VO_Boiler_OT_Enable => VO_Boiler_OT_Enable,
    VO_Boiler_OT_Setpoint => VO_Boiler_OT_Setpoint,
    VO_Boiler_Status => VO_Boiler_Status,
    VO_Any_Subsystem_Degraded => L_Any_Subsystem_Degraded,
    VO_Lead_Boiler => L_Lead_Boiler,
    VO_Demand_Power => L_Demand_Power
);

GVL_STATE.G_Heating_Subsystem_Degraded := L_Any_Subsystem_Degraded;

// >>> BULK_SYNC_ANCHOR: FB_Heating_System_Manager <<<
          
END_FUNCTION_BLOCK

FUNCTION_BLOCK FB_Mode_Manager
  VAR_INPUT
    VI_Is_Night : BOOL;
    VI_Away_Request : BOOL;
    VI_Maintenance_Request : BOOL;
    VI_System_Time_MS : UDINT;
  END_VAR
  VAR_OUTPUT
    VO_Mode : E_Behavior_Mode;
    VO_Mode_Code : UDINT;
  END_VAR

            // default
VO_Mode := BEHAVIOR_HOME;
VO_Mode_Code := 0;

// priority-based transitions
IF VI_Maintenance_Request THEN
    VO_Mode := BEHAVIOR_MAINTENANCE;
    VO_Mode_Code := 300;
ELSIF VI_Away_Request THEN
    VO_Mode := BEHAVIOR_AWAY;
    VO_Mode_Code := 200;
ELSIF VI_Is_Night THEN
    VO_Mode := BEHAVIOR_NIGHT;
    VO_Mode_Code := 100;
END_IF;
          
END_FUNCTION_BLOCK

FUNCTION_BLOCK FB_State_Manager
  VAR_INPUT
    VI_System_Severity : E_System_Severity;
    VI_Root_Cause : E_System_Root_Cause;
    VI_Freeze_Risk : BOOL := FALSE;
  END_VAR
  VAR_OUTPUT
    VO_System_OK : BOOL;
    VO_System_Warning : BOOL;
    VO_System_Critical : BOOL;
    VO_Status_Msg : STRING(200);
    VO_System_Mode : E_System_Operating_Mode;
  END_VAR

            VO_System_OK := FALSE;
VO_System_Warning := FALSE;
VO_System_Critical := FALSE;
VO_Status_Msg := '';
VO_System_Mode := E_System_Operating_Mode.MODE_NORMAL;

CASE VI_System_Severity OF
    E_System_Severity.SEV_NORMAL:
        VO_System_OK := TRUE;
        VO_Status_Msg := 'Система в норме';
        VO_System_Mode := E_System_Operating_Mode.MODE_NORMAL;

    E_System_Severity.SEV_WARNING:
        VO_System_Warning := TRUE;
        VO_System_Mode := E_System_Operating_Mode.MODE_DEGRADED;
        CASE VI_Root_Cause OF
            E_System_Root_Cause.ROOT_WATER_LEAK:
                VO_Status_Msg := 'Предупреждение: протечка воды';
            E_System_Root_Cause.ROOT_CO_WARNING:
                VO_Status_Msg := 'Предупреждение: повышенный CO';
            ELSE
                VO_Status_Msg := 'Предупреждение системы';
        END_CASE;

    E_System_Severity.SEV_DEGRADED:
        VO_System_Warning := TRUE;
        VO_System_Mode := E_System_Operating_Mode.MODE_DEGRADED;
        CASE VI_Root_Cause OF
            E_System_Root_Cause.ROOT_SENSOR_FAULT:
                VO_Status_Msg := 'Деградация: ошибка датчика';
            E_System_Root_Cause.ROOT_IO_OFFLINE:
                VO_Status_Msg := 'Деградация: модуль IO недоступен';
            E_System_Root_Cause.ROOT_COMM_FAULT:
                VO_Status_Msg := 'Деградация: ошибка связи';
            E_System_Root_Cause.ROOT_WATCHDOG_FAULT:
                VO_Status_Msg := 'Деградация: watchdog fault';
            E_System_Root_Cause.ROOT_SUBSYSTEM_FAULT:
                VO_Status_Msg := 'Деградация: ошибка подсистемы';
            ELSE
                VO_Status_Msg := 'Деградация системы';
        END_CASE;

    E_System_Severity.SEV_CRITICAL:
        VO_System_Critical := TRUE;

        IF (VI_Root_Cause = E_System_Root_Cause.ROOT_GAS_LEAK OR
            VI_Root_Cause = E_System_Root_Cause.ROOT_CO_CRITICAL) AND
            VI_Freeze_Risk THEN
            VO_System_Mode := E_System_Operating_Mode.MODE_FREEZE_PROTECTION;
        ELSE
            VO_System_Mode := E_System_Operating_Mode.MODE_SAFE_STOP;
        END_IF;

        CASE VI_Root_Cause OF
            E_System_Root_Cause.ROOT_FIRE:
                VO_Status_Msg := 'АВАРИЯ: ПОЖАР';
            E_System_Root_Cause.ROOT_GAS_LEAK:
                VO_Status_Msg := 'АВАРИЯ: УТЕЧКА ГАЗА';
            E_System_Root_Cause.ROOT_CO_CRITICAL:
                VO_Status_Msg := 'АВАРИЯ: КРИТИЧЕСКИЙ CO';
            E_System_Root_Cause.ROOT_WATCHDOG_FAULT:
                VO_Status_Msg := 'АВАРИЯ: WATCHDOG';
            ELSE
                VO_Status_Msg := 'АВАРИЯ СИСТЕМЫ';
        END_CASE;
END_CASE;
// >>> BULK_SYNC_ANCHOR: FB_State_Manager <<<
          
END_FUNCTION_BLOCK

FUNCTION_BLOCK FB_Heating_Safety_Gate
  VAR_INPUT
    VI_System_Mode : E_System_Operating_Mode;
    VI_Emergency_Stop : BOOL;
    VI_Gas_Safety_Stop : BOOL;
    VI_IO_Failsafe_Active : BOOL;
    VI_Outdoor_Temp : REAL;
    VI_Freeze_Threshold : REAL;
  END_VAR
  VAR_OUTPUT
    VO_Block_Normal_Heating : BOOL;
    VO_Gas_Safety_Active : BOOL;
    VO_Emergency_Safe_Stop_Active : BOOL;
    VO_IO_Failsafe_Active : BOOL;
    VO_Freeze_Mode_Active : BOOL;
    VO_Freeze_Target_Supply : REAL;
  END_VAR
  VAR_IN_OUT
    VI_Floor_Temps : ARRAY[1..GVL_CONSTANTS.C_MAX_HEATING_CIRCUITS] OF REAL;
  END_VAR
  VAR
    L_i : INT;
  END_VAR

            // ==============================================================================
// Heating safety gate helper
//
// Internal helper for FB_Heating_System_Manager.
// Owns common safety/freeze decision calculation. The manager remains the public
// facade and still projects physical safe-state outputs.
// ==============================================================================



VO_Gas_Safety_Active := VI_Gas_Safety_Stop;
VO_Emergency_Safe_Stop_Active := VI_Emergency_Stop OR (VI_System_Mode = E_System_Operating_Mode.MODE_SAFE_STOP);
VO_IO_Failsafe_Active := VI_IO_Failsafe_Active;

VO_Block_Normal_Heating := VO_Gas_Safety_Active OR VO_Emergency_Safe_Stop_Active OR VO_IO_Failsafe_Active;
VO_Freeze_Mode_Active := (VI_System_Mode = E_System_Operating_Mode.MODE_FREEZE_PROTECTION) OR (VI_Outdoor_Temp < -5.0);

FOR L_i := 1 TO GVL_CONSTANTS.C_MAX_HEATING_CIRCUITS DO
    IF VI_Floor_Temps[L_i] < 7.0 THEN
        VO_Freeze_Mode_Active := TRUE;
    END_IF;
END_FOR;

IF VO_Freeze_Mode_Active THEN
    VO_Freeze_Target_Supply := LIMIT(20.0, VI_Freeze_Threshold + 2.0, 35.0);
ELSE
    VO_Freeze_Target_Supply := 0.0;
END_IF;

// >>> BULK_SYNC_ANCHOR: FB_Heating_Safety_Gate <<<
          
END_FUNCTION_BLOCK

FUNCTION_BLOCK FB_Scenario_Transition_Guard
  VAR_INPUT
    VI_Current_Scenario : E_SCENARIO_TYPE;
    VI_Target_Scenario : E_SCENARIO_TYPE;
  END_VAR
  VAR_OUTPUT
    VO_Transition_Allowed : BOOL;
    VO_Reason : STRING(120);
  END_VAR

            VO_Transition_Allowed := TRUE;
VO_Reason := 'OK';

// no-op transition is always allowed
IF VI_Current_Scenario = VI_Target_Scenario THEN
    RETURN;
END_IF;

// emergency can always be entered
IF VI_Target_Scenario = E_SCENARIO_TYPE.SCENARIO_EMERGENCY THEN
    RETURN;
END_IF;

// from NONE, any target is allowed
IF VI_Current_Scenario = E_SCENARIO_TYPE.SCENARIO_NONE THEN
    RETURN;
END_IF;

// emergency exit is restricted
IF VI_Current_Scenario = E_SCENARIO_TYPE.SCENARIO_EMERGENCY THEN
    CASE VI_Target_Scenario OF
        E_SCENARIO_TYPE.SCENARIO_NONE,
        E_SCENARIO_TYPE.SCENARIO_AWAY,
        E_SCENARIO_TYPE.SCENARIO_SLEEP,
        E_SCENARIO_TYPE.SCENARIO_PRESENCE:
            RETURN;
    ELSE
        VO_Transition_Allowed := FALSE;
        VO_Reason := 'Переход из EMERGENCY в данный сценарий запрещён';
        RETURN;
    END_CASE;
END_IF;

// away exit is restricted to safe occupancy contexts
IF VI_Current_Scenario = E_SCENARIO_TYPE.SCENARIO_AWAY THEN
    CASE VI_Target_Scenario OF
        E_SCENARIO_TYPE.SCENARIO_NONE,
        E_SCENARIO_TYPE.SCENARIO_SLEEP,
        E_SCENARIO_TYPE.SCENARIO_PRESENCE,
        E_SCENARIO_TYPE.SCENARIO_EMERGENCY:
            RETURN;
    ELSE
        VO_Transition_Allowed := FALSE;
        VO_Reason := 'Переход из AWAY в данный сценарий запрещён';
        RETURN;
    END_CASE;
END_IF;

// default: allow
RETURN;
// >>> BULK_SYNC_ANCHOR: FB_Scenario_Transition_Guard <<<
          
END_FUNCTION_BLOCK

FUNCTION_BLOCK FB_Alarm_Manager
  VAR_INPUT
    VI_System_Time_MS : UDINT;
    VI_IsActivePLC : BOOL;
    VI_Gas_Alarm : BOOL;
    VI_Fire_Alarm : BOOL;
    VI_Flood_Alarm : BOOL;
    VI_Security_Alarm : BOOL;
    VI_First_Fault_Active : BOOL;
    VI_First_Fault_Type : INT;
    VI_First_Fault_Source : INT;
    VI_Security_Msg : STRING(200);
    VI_Acknowledge_All : BOOL;
    VI_Mute_Siren : BOOL;
  END_VAR
  VAR_OUTPUT
    VO_Global_Critical : BOOL;
    VO_Global_Warning : BOOL;
    VO_Siren_Active : BOOL;
    VO_Active_Count : INT;
    VO_Unacked_Count : INT;
    VO_Event_Pulse : BOOL;
    VO_Event_Code : UDINT;
    VO_Event_Value : REAL;
    VO_Alarm_List : ARRAY[1..GVL_CONSTANTS.C_MAX_ALARMS] OF ST_Alarm_Record;
  END_VAR
  VAR_IN_OUT
    VI_Boiler_Errors : ARRAY[1..GVL_CONSTANTS.C_MAX_BOILERS] OF BOOL;
  END_VAR
  VAR_IN_OUT
    VIO_Next_Alarm_ID : UDINT;
  END_VAR
  VAR
    L_i, L_j, L_k : INT;
    L_Target_Slot : INT;
    L_Min_Pri : INT;
    L_Pending_Alarms : ARRAY[1..10] OF ST_Alarm_Record;
    L_Pending_Count : INT := 0;
    T_Debounce_Gas : FB_System_Timer;
    T_Debounce_Fire : FB_System_Timer;
    T_Debounce_Flood : FB_System_Timer;
    T_Debounce_Security : FB_System_Timer;
    R_Trig_Gas : R_TRIG;
    R_Trig_Fire : R_TRIG;
    R_Trig_Flood : R_TRIG;
    R_Trig_Security : R_TRIG;
    R_Trig_First_Fault : R_TRIG;
    R_Trig_Boiler : ARRAY[1..GVL_CONSTANTS.C_MAX_BOILERS] OF R_TRIG;
    L_First_Fault_Source_Text : STRING(32);
    L_First_Fault_Type_Text : STRING(32);
    L_Event_Pulse_Latched : BOOL;
  END_VAR

            VO_Event_Pulse := FALSE;
VO_Event_Code := 0;
VO_Event_Value := 0.0;

// 1. Детекция новых тревог (антидребезг + передний фронт)
T_Debounce_Gas(IN := VI_Gas_Alarm, PT := T#100ms, VI_System_Time_MS := VI_System_Time_MS);
T_Debounce_Fire(IN := VI_Fire_Alarm, PT := T#100ms, VI_System_Time_MS := VI_System_Time_MS);
T_Debounce_Flood(IN := VI_Flood_Alarm, PT := T#500ms, VI_System_Time_MS := VI_System_Time_MS);
T_Debounce_Security(IN := VI_Security_Alarm, PT := T#100ms, VI_System_Time_MS := VI_System_Time_MS);

R_Trig_Gas(CLK := T_Debounce_Gas.Q);
R_Trig_Fire(CLK := T_Debounce_Fire.Q);
R_Trig_Flood(CLK := T_Debounce_Flood.Q);
R_Trig_Security(CLK := T_Debounce_Security.Q);
R_Trig_First_Fault(CLK := VI_First_Fault_Active);
FOR L_i := 1 TO GVL_CONSTANTS.C_MAX_BOILERS DO
    R_Trig_Boiler[L_i](CLK := VI_Boiler_Errors[L_i]);
END_FOR;

// 2. Добавление новых тревог в список (Кольцевой буфер)
L_Pending_Count := 0;
L_Event_Pulse_Latched := FALSE;

IF R_Trig_Gas.Q AND L_Pending_Count < 10 THEN
    L_Pending_Count := L_Pending_Count + 1;
    L_Pending_Alarms[L_Pending_Count].Timestamp_MS := VI_System_Time_MS;
    L_Pending_Alarms[L_Pending_Count].Source := 'Gas';
    L_Pending_Alarms[L_Pending_Count].Source_ID := 0;
    L_Pending_Alarms[L_Pending_Count].Message := 'Критическая концентрация газа!';
    L_Pending_Alarms[L_Pending_Count].Severity := E_ALERT_PRIORITY.ALERT_PRIORITY_CRITICAL;
    L_Pending_Alarms[L_Pending_Count].Is_Active := TRUE;
    L_Pending_Alarms[L_Pending_Count].Is_Acknowledged := FALSE;
END_IF;

IF R_Trig_Fire.Q AND L_Pending_Count < 10 THEN
    L_Pending_Count := L_Pending_Count + 1;
    L_Pending_Alarms[L_Pending_Count].Timestamp_MS := VI_System_Time_MS;
    L_Pending_Alarms[L_Pending_Count].Source := 'Fire';
    L_Pending_Alarms[L_Pending_Count].Source_ID := 0;
    L_Pending_Alarms[L_Pending_Count].Message := 'Обнаружено задымление!';
    L_Pending_Alarms[L_Pending_Count].Severity := E_ALERT_PRIORITY.ALERT_PRIORITY_CRITICAL;
    L_Pending_Alarms[L_Pending_Count].Is_Active := TRUE;
    L_Pending_Alarms[L_Pending_Count].Is_Acknowledged := FALSE;
END_IF;

IF R_Trig_Flood.Q AND L_Pending_Count < 10 THEN
    L_Pending_Count := L_Pending_Count + 1;
    L_Pending_Alarms[L_Pending_Count].Timestamp_MS := VI_System_Time_MS;
    L_Pending_Alarms[L_Pending_Count].Source := 'Flood';
    L_Pending_Alarms[L_Pending_Count].Source_ID := 0;
    L_Pending_Alarms[L_Pending_Count].Message := 'Обнаружена протечка воды!';
    L_Pending_Alarms[L_Pending_Count].Severity := E_ALERT_PRIORITY.ALERT_PRIORITY_CRITICAL;
    L_Pending_Alarms[L_Pending_Count].Is_Active := TRUE;
    L_Pending_Alarms[L_Pending_Count].Is_Acknowledged := FALSE;
END_IF;

IF R_Trig_Security.Q AND L_Pending_Count < 10 THEN
    L_Pending_Count := L_Pending_Count + 1;
    L_Pending_Alarms[L_Pending_Count].Timestamp_MS := VI_System_Time_MS;
    L_Pending_Alarms[L_Pending_Count].Source := 'Security';
    L_Pending_Alarms[L_Pending_Count].Source_ID := 0;
    L_Pending_Alarms[L_Pending_Count].Message := VI_Security_Msg;
    L_Pending_Alarms[L_Pending_Count].Severity := E_ALERT_PRIORITY.ALERT_PRIORITY_CRITICAL;
    L_Pending_Alarms[L_Pending_Count].Is_Active := TRUE;
    L_Pending_Alarms[L_Pending_Count].Is_Acknowledged := FALSE;
END_IF;

IF R_Trig_First_Fault.Q AND L_Pending_Count < 10 THEN
    L_Pending_Count := L_Pending_Count + 1;
    L_Pending_Alarms[L_Pending_Count].Timestamp_MS := VI_System_Time_MS;
    L_Pending_Alarms[L_Pending_Count].Source := 'Diagnostics';
    L_Pending_Alarms[L_Pending_Count].Source_ID := TO_BYTE(VI_First_Fault_Source);

    CASE VI_First_Fault_Type OF
        1: L_First_Fault_Type_Text := 'IO';
        2: L_First_Fault_Type_Text := 'Sensor';
        3: L_First_Fault_Type_Text := 'Comm';
        4: L_First_Fault_Type_Text := 'Subsystem';
        ELSE L_First_Fault_Type_Text := 'Unknown';
    END_CASE;

    CASE VI_First_Fault_Source OF
        1: L_First_Fault_Source_Text := 'Heating';
        2: L_First_Fault_Source_Text := 'DHW';
        3: L_First_Fault_Source_Text := 'Ventilation';
        4: L_First_Fault_Source_Text := 'Lighting';
        5: L_First_Fault_Source_Text := 'Access';
        ELSE L_First_Fault_Source_Text := 'Unknown';
    END_CASE;

    L_Pending_Alarms[L_Pending_Count].Message := CONCAT('Diagnostics root cause: ', CONCAT(L_First_Fault_Source_Text, CONCAT(' / ', L_First_Fault_Type_Text)));
    L_Pending_Alarms[L_Pending_Count].Severity := E_ALERT_PRIORITY.ALERT_PRIORITY_HIGH;
    L_Pending_Alarms[L_Pending_Count].Is_Active := TRUE;
    L_Pending_Alarms[L_Pending_Count].Is_Acknowledged := FALSE;
END_IF;

FOR L_j := 1 TO GVL_CONSTANTS.C_MAX_BOILERS DO
    IF R_Trig_Boiler[L_j].Q AND L_Pending_Count < 10 THEN
        L_Pending_Count := L_Pending_Count + 1;
        L_Pending_Alarms[L_Pending_Count].Timestamp_MS := VI_System_Time_MS;
        L_Pending_Alarms[L_Pending_Count].Source := 'Boiler';
        L_Pending_Alarms[L_Pending_Count].Source_ID := TO_BYTE(L_j);
        L_Pending_Alarms[L_Pending_Count].Message := CONCAT('Авария котла №', INT_TO_STRING(L_j));
        L_Pending_Alarms[L_Pending_Count].Severity := E_ALERT_PRIORITY.ALERT_PRIORITY_HIGH;
        L_Pending_Alarms[L_Pending_Count].Is_Active := TRUE;
        L_Pending_Alarms[L_Pending_Count].Is_Acknowledged := FALSE;
    END_IF;
END_FOR;



// Обработка очереди новых тревог с учетом приоритетов
FOR L_i := 1 TO L_Pending_Count DO

    L_Target_Slot := 0;
    
    // 1. Ищем пустой слот
    FOR L_k := 1 TO GVL_CONSTANTS.C_MAX_ALARMS DO
        IF VO_Alarm_List[L_k].ID = 0 THEN
            L_Target_Slot := L_k;
            EXIT;
        END_IF;
    END_FOR;
    
    // 2. Ищем квитированную тревогу с наименьшим приоритетом
    IF L_Target_Slot = 0 THEN
        L_Min_Pri := 999;
        FOR L_k := 1 TO GVL_CONSTANTS.C_MAX_ALARMS DO
            IF VO_Alarm_List[L_k].Is_Acknowledged AND TO_INT(VO_Alarm_List[L_k].Severity) < L_Min_Pri THEN
                L_Min_Pri := TO_INT(VO_Alarm_List[L_k].Severity);
                L_Target_Slot := L_k;
            END_IF;
        END_FOR;
    END_IF;
    
    // 3. Ищем неквитированную тревогу с наименьшим приоритетом (если он ниже добавляемой)
    IF L_Target_Slot = 0 THEN
        L_Min_Pri := 999;
        FOR L_k := 1 TO GVL_CONSTANTS.C_MAX_ALARMS DO
            IF TO_INT(VO_Alarm_List[L_k].Severity) < L_Min_Pri AND TO_INT(VO_Alarm_List[L_k].Severity) < TO_INT(L_Pending_Alarms[L_i].Severity) THEN
                L_Min_Pri := TO_INT(VO_Alarm_List[L_k].Severity);
                L_Target_Slot := L_k;
            END_IF;
        END_FOR;
    END_IF;
    
    IF L_Target_Slot = 0 THEN 
        // Буфер полон критических неквитированных тревог. Не затираем!
        CONTINUE; 
    END_IF;
    
    VO_Alarm_List[L_Target_Slot] := L_Pending_Alarms[L_i];
    VO_Alarm_List[L_Target_Slot].ID := VIO_Next_Alarm_ID;
    VIO_Next_Alarm_ID := VIO_Next_Alarm_ID + 1;
    IF VIO_Next_Alarm_ID = 0 THEN VIO_Next_Alarm_ID := 1; END_IF;
    IF NOT L_Event_Pulse_Latched THEN
        VO_Event_Pulse := TRUE;
        VO_Event_Code := 1203;
        VO_Event_Value := TO_REAL(VO_Alarm_List[L_Target_Slot].Severity);
        L_Event_Pulse_Latched := TRUE;
    END_IF;
END_FOR;

// 3. Обновление статуса существующих тревог (ушли ли они?)
FOR L_i := 1 TO GVL_CONSTANTS.C_MAX_ALARMS DO
    IF VO_Alarm_List[L_i].ID <> 0 THEN
        IF VO_Alarm_List[L_i].Source = 'Gas' THEN VO_Alarm_List[L_i].Is_Active := VI_Gas_Alarm;
        ELSIF VO_Alarm_List[L_i].Source = 'Fire' THEN VO_Alarm_List[L_i].Is_Active := VI_Fire_Alarm;
        ELSIF VO_Alarm_List[L_i].Source = 'Flood' THEN VO_Alarm_List[L_i].Is_Active := VI_Flood_Alarm;
        ELSIF VO_Alarm_List[L_i].Source = 'Security' THEN VO_Alarm_List[L_i].Is_Active := VI_Security_Alarm;
        ELSIF VO_Alarm_List[L_i].Source = 'Diagnostics' THEN VO_Alarm_List[L_i].Is_Active := VI_First_Fault_Active;
        ELSIF VO_Alarm_List[L_i].Source = 'Boiler' THEN 
            IF TO_INT(VO_Alarm_List[L_i].Source_ID) >= 1 AND TO_INT(VO_Alarm_List[L_i].Source_ID) <= GVL_CONSTANTS.C_MAX_BOILERS THEN
                VO_Alarm_List[L_i].Is_Active := VI_Boiler_Errors[TO_INT(VO_Alarm_List[L_i].Source_ID)];
            END_IF;
        END_IF;
    END_IF;
END_FOR;

// 4. Квитирование тревог
IF VI_Acknowledge_All THEN
    FOR L_i := 1 TO GVL_CONSTANTS.C_MAX_ALARMS DO
        IF VO_Alarm_List[L_i].ID <> 0 THEN
            VO_Alarm_List[L_i].Is_Acknowledged := TRUE;
        END_IF;
    END_FOR;

    IF NOT L_Event_Pulse_Latched THEN
        VO_Event_Pulse := TRUE;
        VO_Event_Code := 1201;
        VO_Event_Value := TO_REAL(VO_Unacked_Count);
        L_Event_Pulse_Latched := TRUE;
    END_IF;
END_IF;

// 4.5 Автоквитирование некритичных тревог, если они больше не активны
FOR L_i := 1 TO GVL_CONSTANTS.C_MAX_ALARMS DO
    IF VO_Alarm_List[L_i].ID <> 0 AND NOT VO_Alarm_List[L_i].Is_Active AND NOT VO_Alarm_List[L_i].Is_Acknowledged THEN
        IF VO_Alarm_List[L_i].Severity <> E_ALERT_PRIORITY.ALERT_PRIORITY_CRITICAL THEN
            VO_Alarm_List[L_i].Is_Acknowledged := TRUE;
        END_IF;
    END_IF;
END_FOR;

// 5. Очистка списка (удаление неактивных И квитированных тревог)
// В кольцевом буфере мы просто помечаем слот как пустой (ID = 0), без сдвига массива
FOR L_i := 1 TO GVL_CONSTANTS.C_MAX_ALARMS DO
    IF VO_Alarm_List[L_i].ID <> 0 AND NOT VO_Alarm_List[L_i].Is_Active AND VO_Alarm_List[L_i].Is_Acknowledged THEN
        // Удаляем тревогу
        VO_Alarm_List[L_i].ID := 0;
        IF NOT L_Event_Pulse_Latched THEN
            VO_Event_Pulse := TRUE;
            VO_Event_Code := 1202;
            VO_Event_Value := 0.0;
            L_Event_Pulse_Latched := TRUE;
        END_IF;
    END_IF;
END_FOR;


// 6. Подсчет статистики и формирование глобальных флагов
VO_Global_Critical := FALSE;
VO_Global_Warning := FALSE;
VO_Siren_Active := FALSE;
VO_Active_Count := 0;
VO_Unacked_Count := 0;

FOR L_i := 1 TO GVL_CONSTANTS.C_MAX_ALARMS DO
    IF VO_Alarm_List[L_i].ID <> 0 THEN
        IF VO_Alarm_List[L_i].Is_Active THEN
            VO_Active_Count := VO_Active_Count + 1;
        END_IF;
        
        IF NOT VO_Alarm_List[L_i].Is_Acknowledged THEN
            VO_Unacked_Count := VO_Unacked_Count + 1;
            
            IF VO_Alarm_List[L_i].Severity = E_ALERT_PRIORITY.ALERT_PRIORITY_CRITICAL THEN
                VO_Global_Critical := TRUE;
                // Сирена работает только для неквитированных критических тревог, если не включен Mute
                IF NOT VI_Mute_Siren THEN
                    VO_Siren_Active := TRUE;
                END_IF;
            ELSIF VO_Alarm_List[L_i].Severity = E_ALERT_PRIORITY.ALERT_PRIORITY_HIGH THEN
                VO_Global_Warning := TRUE;
            END_IF;
        END_IF;
    END_IF;
END_FOR;
// >>> BULK_SYNC_ANCHOR: FB_Alarm_Manager <<<
          
END_FUNCTION_BLOCK

FUNCTION_BLOCK FB_Presence_Playback
  VAR_INPUT
    VI_Mode_Record : BOOL;
    VI_Time_Index : UDINT;
  END_VAR
  VAR_OUTPUT
    VO_Light_Outputs : ARRAY[1..32] OF BOOL;
  END_VAR
  VAR_IN_OUT
    VI_Light_Inputs : ARRAY[1..32] OF BOOL;
  END_VAR
  VAR
    L_Current_Slot : UDINT;
    L_i : INT;
  END_VAR

            L_Current_Slot := (VI_Time_Index / (GVL_CONSTANTS.C_MS_IN_MINUTE * 10)) MOD TO_UDINT(GVL_CONSTANTS.C_MAX_PRESENCE_HISTORY); // Слот каждые 10 минут

IF VI_Mode_Record THEN
    // Запись текущего состояния в слот
    GVL_Retain.G_Presence_History[L_Current_Slot] := 0;
    FOR L_i := 1 TO 32 DO
        IF VI_Light_Inputs[L_i] THEN
            GVL_Retain.G_Presence_History[L_Current_Slot] := GVL_Retain.G_Presence_History[L_Current_Slot] OR SHL(WORD#1, L_i-1);
        END_IF;
    END_FOR;
ELSE
    // Воспроизведение из слота
    FOR L_i := 1 TO 32 DO
        VO_Light_Outputs[L_i] := (GVL_Retain.G_Presence_History[L_Current_Slot] AND SHL(WORD#1, L_i-1)) <> 0;
    END_FOR;
END_IF;
          
END_FUNCTION_BLOCK

FUNCTION_BLOCK FB_Random_Generator
  VAR_INPUT
    VI_Seed_Value : UDINT;
  END_VAR
  VAR_INPUT
    VI_min : UDINT;
    VI_max : UDINT;
    VI_System_Time_MS : UDINT;
  END_VAR
  VAR
    L_seed : UDINT := 1;
    L_Is_Seeded : BOOL := FALSE;
  END_VAR
  VAR CONSTANT
    C_LCG_MULTIPLIER : UDINT := 1664525;
    C_LCG_INCREMENT : UDINT := 1013904223;
    C_LCG_MODULUS : LREAL := 4294967296.0;
  END_VAR
  VAR
    L_range : UDINT;
    L_rand_factor : LREAL;
  END_VAR

            METHOD Seed : BOOL

L_seed := VI_Seed_Value;
L_Is_Seeded := TRUE;
Seed := TRUE;
END_METHOD

METHOD Random_Int_Range : UDINT


IF NOT L_Is_Seeded AND VI_System_Time_MS > 0 THEN
    L_seed := VI_System_Time_MS;
    L_Is_Seeded := TRUE;
END_IF;

L_seed := (C_LCG_MULTIPLIER * L_seed) + C_LCG_INCREMENT;

IF VI_max > VI_min THEN
        L_range := VI_max - VI_min;
        // Используем LREAL для точности и исключения выхода за границу
        L_rand_factor := TO_LREAL(L_seed) / C_LCG_MODULUS;
        Random_Int_Range := VI_min + TO_UDINT(L_rand_factor * TO_LREAL(L_range + 1));
        
        // Финальная защита от переполнения
        IF Random_Int_Range > VI_max THEN
            Random_Int_Range := VI_max;
        END_IF;
    ELSE
        Random_Int_Range := VI_min;
    END_IF;
          
END_FUNCTION_BLOCK

FUNCTION_BLOCK FB_Ventilation_System_Manager
  VAR_INPUT
    VI_System_Time_MS : UDINT;
    VI_IsActivePLC : BOOL;
    VI_Outdoor_Temp : REAL;
    VI_Current_Scenario : E_SCENARIO_TYPE;
    VI_System_Mode : E_System_Operating_Mode;
    VI_Config : ST_Ventilation_Global_Config;
    VI_Fire_Alarm : BOOL;
    VI_Gas_Alarm : BOOL;
    VI_PV3_Boost_Req : BOOL;
    VI_Supply_100_Req : BOOL;
    VI_Exhaust_100_Req : BOOL;
    VI_Supply_80_Req : BOOL;
    VI_Vent_Stop : BOOL;
    VI_IO_Modules_Online : ARRAY[1..GVL_CONSTANTS.C_MAX_MODULES] OF BOOL;
  END_VAR
  VAR_OUTPUT
    VO_Supply_Fans : ARRAY[1..GVL_CONSTANTS.C_MAX_SUPPLY_FANS] OF BYTE;
    VO_Exhaust_Fans : ARRAY[1..GVL_CONSTANTS.C_MAX_EXHAUST_FANS] OF BYTE;
    VO_Heater_Power : ARRAY[1..GVL_CONSTANTS.C_MAX_BOILERS] OF REAL;
    VO_Status_Msg : STRING(200);
    VO_Ventilation_IO_Fault : BOOL;
    VO_Ventilation_Subsystem_Degraded : BOOL;
  END_VAR
  VAR_IN_OUT
    VI_Supply_Temps : ARRAY[1..GVL_CONSTANTS.C_MAX_SUPPLY_TEMPS] OF REAL;
    VI_Room_Temps : ARRAY[1..16] OF REAL;
    VI_Room_Humidities : ARRAY[1..16] OF REAL;
    VI_Room_CO2 : ARRAY[1..16] OF REAL;
    VI_Wet_Zone_Active : ARRAY[1..GVL_CONSTANTS.C_MAX_WET_ZONES] OF BOOL;
    VI_Rule_Actions : ARRAY[1..GVL_CONSTANTS.C_MAX_RULES] OF ST_Rule_Action;
  END_VAR
  VAR
    L_Policy_Normal : BOOL;
    L_Policy_Safe_Stop : BOOL;
    L_Policy_Degraded : BOOL;
    L_Policy_Freeze_Protection : BOOL;
    L_i : INT;
    L_j : INT;
    L_Max_CO2 : REAL;
    L_Max_Hum : REAL;
    L_Base_Speed : BYTE;
    L_Target_Temp : REAL;
    L_PID_Heaters : ARRAY[1..GVL_CONSTANTS.C_MAX_BOILERS] OF FB_PID_Controller;
    L_Wet_Zone_Timers : ARRAY[1..GVL_CONSTANTS.C_MAX_WET_ZONES] OF FB_System_Timer_TOF;
  END_VAR

            // ========================================
// Ventilation policy layer
// ========================================
VO_Ventilation_IO_Fault := FALSE;
VO_Ventilation_Subsystem_Degraded := FALSE;
L_Policy_Normal := (VI_System_Mode = E_System_Operating_Mode.MODE_NORMAL);
L_Policy_Safe_Stop := (VI_System_Mode = E_System_Operating_Mode.MODE_SAFE_STOP);
L_Policy_Degraded := (VI_System_Mode = E_System_Operating_Mode.MODE_DEGRADED);
L_Policy_Freeze_Protection := (VI_System_Mode = E_System_Operating_Mode.MODE_FREEZE_PROTECTION);

IF NOT VI_IsActivePLC THEN
    FOR L_i := 1 TO GVL_CONSTANTS.C_MAX_SUPPLY_FANS DO
        VO_Supply_Fans[L_i] := 0;
        IF L_i <= GVL_CONSTANTS.C_MAX_SUPPLY_TEMPS THEN
            VO_Heater_Power[L_i] := 0.0;
        END_IF;
    END_FOR;
    FOR L_i := 1 TO GVL_CONSTANTS.C_MAX_EXHAUST_FANS DO
        VO_Exhaust_Fans[L_i] := 0;
    END_FOR;
    VO_Status_Msg := 'ВЕНТИЛЯЦИЯ: РЕЗЕРВНЫЙ ПЛК';
    RETURN;
END_IF;

// Проверка связи с модулями ввода-вывода
FOR L_i := 1 TO GVL_CONSTANTS.C_MAX_MODULES DO
    IF NOT VI_IO_Modules_Online[L_i] THEN
        VO_Ventilation_IO_Fault := TRUE;
        // Переход в безопасное состояние при потере связи (отключение вентиляции)
        FOR L_j := 1 TO GVL_CONSTANTS.C_MAX_SUPPLY_FANS DO
            VO_Supply_Fans[L_j] := 0;
        END_FOR;
        FOR L_j := 1 TO GVL_CONSTANTS.C_MAX_EXHAUST_FANS DO
            VO_Exhaust_Fans[L_j] := 0;
        END_FOR;
        FOR L_j := 1 TO GVL_CONSTANTS.C_MAX_BOILERS DO
            VO_Heater_Power[L_j] := 0.0;
        END_FOR;
        VO_Status_Msg := 'ОШИБКА: Потеря связи с модулями ввода-вывода';
        RETURN;
    END_IF;
END_FOR;

// =========================
// SYSTEM MODE OVERRIDE
// =========================
// VENT_POLICY_ROUTING_PHASE3_V2
IF L_Policy_Safe_Stop THEN
    FOR L_i := 1 TO GVL_CONSTANTS.C_MAX_SUPPLY_FANS DO
        VO_Supply_Fans[L_i] := 0;
    END_FOR;
    FOR L_i := 1 TO GVL_CONSTANTS.C_MAX_EXHAUST_FANS DO
        VO_Exhaust_Fans[L_i] := 0;
    END_FOR;
    FOR L_i := 1 TO GVL_CONSTANTS.C_MAX_BOILERS DO
        VO_Heater_Power[L_i] := 0.0;
    END_FOR;
    VO_Status_Msg := 'ВЕНТИЛЯЦИЯ: ОСТАНОВЛЕНА POLICY SAFE_STOP';
    RETURN;
END_IF;

IF L_Policy_Degraded THEN
    FOR L_i := 1 TO GVL_CONSTANTS.C_MAX_SUPPLY_FANS DO
        VO_Supply_Fans[L_i] := 0;
    END_FOR;
    FOR L_i := 1 TO GVL_CONSTANTS.C_MAX_BOILERS DO
        VO_Heater_Power[L_i] := 0.0;
    END_FOR;
    VO_Ventilation_Subsystem_Degraded := TRUE;
    VO_Status_Msg := 'ВЕНТИЛЯЦИЯ: DEGRADED POLICY';
END_IF;

IF L_Policy_Freeze_Protection THEN
    FOR L_i := 1 TO GVL_CONSTANTS.C_MAX_SUPPLY_FANS DO
        VO_Supply_Fans[L_i] := 0;
    END_FOR;
    FOR L_i := 1 TO GVL_CONSTANTS.C_MAX_EXHAUST_FANS DO
        VO_Exhaust_Fans[L_i] := 0;
    END_FOR;
    FOR L_i := 1 TO GVL_CONSTANTS.C_MAX_BOILERS DO
        VO_Heater_Power[L_i] := 0.0;
    END_FOR;
    VO_Status_Msg := 'ВЕНТИЛЯЦИЯ: FREEZE_PROTECTION POLICY (stop)';
    RETURN;
END_IF;

// MODE_FREEZE_PROTECTION пока оставляем на текущей штатной логике

// 1. Определение базовой скорости и целевой температуры по сценарию (ТЗ 7.1)
CASE VI_Current_Scenario OF
    E_SCENARIO_TYPE.SCENARIO_AWAY:
        L_Base_Speed := VI_Config.Scenario_Modes[3].Base_Fan_Speed;
        L_Target_Temp := VI_Config.Scenario_Modes[3].Target_Temp;
    E_SCENARIO_TYPE.SCENARIO_SLEEP:
        L_Base_Speed := VI_Config.Scenario_Modes[2].Base_Fan_Speed;
        L_Target_Temp := VI_Config.Scenario_Modes[2].Target_Temp;
    ELSE // PRESENCE, MORNING, EVENING
        L_Base_Speed := VI_Config.Scenario_Modes[1].Base_Fan_Speed;
        L_Target_Temp := VI_Config.Scenario_Modes[1].Target_Temp;
END_CASE;

// 2. Логика управления приточными установками (П-1, П-2, П-3)
FOR L_i := 1 TO GVL_CONSTANTS.C_MAX_SUPPLY_FANS DO
    // ПИД-регулирование мощности электрического калорифера
    IF L_i <= GVL_CONSTANTS.C_MAX_SUPPLY_TEMPS THEN
        L_PID_Heaters[L_i](
            VI_SetPoint := L_Target_Temp,
            VI_ProcessValue := VI_Supply_Temps[L_i], // Используем датчик температуры после калорифера
            VI_Kp := 4.0, VI_Tn := 120.0, VI_Tv := 0.0,
            VI_Y_Min := 0.0, VI_Y_Max := 100.0, VI_Cycle_Time_S := 1.0,
            VO_Output => VO_Heater_Power[L_i]
        );
    END_IF;

    // Определение скорости приточного вентилятора
    VO_Supply_Fans[L_i] := L_Base_Speed;
    
    // Обработка действий от Rule Engine
    FOR L_j := 1 TO GVL_CONSTANTS.C_MAX_RULES DO
        IF VI_Rule_Actions[L_j].Active AND VI_Rule_Actions[L_j].Target_ID = L_i THEN
            IF VI_Rule_Actions[L_j].Action_Type = E_Rule_Action_Type.ACTION_SET_VENTILATION THEN
                VO_Supply_Fans[L_i] := REAL_TO_BYTE(VI_Rule_Actions[L_j].Value);
            END_IF;
        END_IF;
    END_FOR;
    
    // Requests are operational requests and must not be reported as subsystem degradation.
END_FOR;

// 3. Логика управления вытяжными установками (В-1 .. В-5)
FOR L_i := 1 TO GVL_CONSTANTS.C_MAX_EXHAUST_FANS DO
    VO_Exhaust_Fans[L_i] := L_Base_Speed;
    
    // ТЗ 4.0: Логика вытяжки в санузлах
    FOR L_j := 1 TO GVL_CONSTANTS.C_MAX_WET_ZONES DO
        IF VI_Config.wet_zone_to_exhaust_map[L_j] = L_i THEN
            // Включение по свету, выключение с задержкой 5 минут (используем TOF)
            L_Wet_Zone_Timers[L_j](IN := VI_Wet_Zone_Active[L_j], PT := T#5m, VI_System_Time_MS := VI_System_Time_MS);
            IF VI_Wet_Zone_Active[L_j] THEN
                VO_Exhaust_Fans[L_i] := 80; // Повышенная скорость при присутствии
            ELSIF L_Wet_Zone_Timers[L_j].Q THEN
                VO_Exhaust_Fans[L_i] := 50; // Скорость выбега (пока таймер TOF активен)
            END_IF;
        END_IF;
    END_FOR;

    // Requests are operational requests and must not be reported as subsystem degradation.
END_FOR;








// ========================================
// VENT_FINAL_CLAMP
// ========================================
IF L_Policy_Degraded THEN
    FOR L_i := 1 TO GVL_CONSTANTS.C_MAX_EXHAUST_FANS DO
        VO_Exhaust_Fans[L_i] := MIN(VO_Exhaust_Fans[L_i], VI_Config.Degraded_Exhaust_Limit);
    END_FOR;
END_IF;

// 4. Формирование статусного сообщения
IF L_Policy_Safe_Stop THEN
    VO_Status_Msg := 'ВЕНТИЛЯЦИЯ: ОСТАНОВЛЕНА POLICY SAFE_STOP';
ELSIF L_Policy_Freeze_Protection THEN
    VO_Status_Msg := 'ВЕНТИЛЯЦИЯ: FREEZE_PROTECTION POLICY (stop)';
ELSIF L_Policy_Degraded THEN
    VO_Status_Msg := 'ВЕНТИЛЯЦИЯ: DEGRADED POLICY';
ELSE
    VO_Status_Msg := 'Вентиляция работает в штатном режиме';
END_IF;
// >>> BULK_SYNC_ANCHOR: FB_Ventilation_System_Manager <<<
          
END_FUNCTION_BLOCK

FUNCTION_BLOCK FB_Device_Predictive_Diag
  VAR_INPUT
    VI_Current_Value : REAL;
    VI_Nominal_Value : REAL;
    VI_Is_Running : BOOL;
    VI_Reset_Stats : BOOL;
    VI_System_Time_MS : UDINT;
  END_VAR
  VAR_IN_OUT
    VIO_Health_Data : ST_Device_Health;
  END_VAR
  VAR
    L_Prev_Running : BOOL;
    L_Start_Time : UDINT;
    L_Last_Calc_Time : UDINT;
    L_Elapsed_MS : UDINT;
    L_Accumulated_MS : UDINT;
    L_Timer_Running : FB_System_Timer;
  END_VAR

            // 0. Сброс статистики
IF VI_Reset_Stats THEN
    VIO_Health_Data.Starts_Count := 0;
    VIO_Health_Data.Sample_Count := 0;
    VIO_Health_Data.Current_Sum := 0.0;
    VIO_Health_Data.Avg_Start_Current := 0.0;
    VIO_Health_Data.Health_Score := 100;
    VIO_Health_Data.Maintenance_Required := FALSE;
    VIO_Health_Data.Warning_Message := '';
    VIO_Health_Data.Last_Start_Current := 0.0;
    VIO_Health_Data.Total_Runtime_Hours := 0;
    L_Accumulated_MS := 0;
END_IF;

// 1. Счётчик пусков и замер пускового тока
IF VI_Is_Running AND NOT L_Prev_Running THEN
    VIO_Health_Data.Starts_Count := VIO_Health_Data.Starts_Count + 1;
    VIO_Health_Data.Last_Start_Current := VI_Current_Value;
    L_Start_Time := VI_System_Time_MS;
    L_Last_Calc_Time := VI_System_Time_MS;
    
    // Обновление среднего пускового тока
    VIO_Health_Data.Sample_Count := VIO_Health_Data.Sample_Count + 1;
    VIO_Health_Data.Current_Sum := VIO_Health_Data.Current_Sum + VI_Current_Value;
    VIO_Health_Data.Avg_Start_Current := VIO_Health_Data.Current_Sum / UDINT_TO_REAL(VIO_Health_Data.Sample_Count);
    
    // 2. Анализ отклонения пускового тока (п. 12.1 ТЗ)
    IF VI_Current_Value > (VI_Nominal_Value * 1.5) THEN
        VIO_Health_Data.Health_Score := TO_BYTE(LIMIT(0, TO_INT(VIO_Health_Data.Health_Score) - 5, 100));
    ELSIF VI_Current_Value > (VI_Nominal_Value * 1.2) THEN
        VIO_Health_Data.Health_Score := TO_BYTE(LIMIT(0, TO_INT(VIO_Health_Data.Health_Score) - 1, 100));
    ELSIF VI_Current_Value < (VI_Nominal_Value * 0.5) THEN
        VIO_Health_Data.Health_Score := TO_BYTE(LIMIT(0, TO_INT(VIO_Health_Data.Health_Score) - 2, 100));
    END_IF;
END_IF;

// 3. Анализ рабочего тока и наработки
IF VI_Is_Running THEN
    L_Elapsed_MS := (VI_System_Time_MS - L_Last_Calc_Time);
    L_Accumulated_MS := L_Accumulated_MS + L_Elapsed_MS;
    L_Last_Calc_Time := VI_System_Time_MS;
    
    // Обновляем наработку каждый час (3600000 мс)
    IF L_Accumulated_MS >= 3600000 THEN
        VIO_Health_Data.Total_Runtime_Hours := VIO_Health_Data.Total_Runtime_Hours + 1;
        L_Accumulated_MS := L_Accumulated_MS - 3600000;
        
        // Естественный износ: -1% здоровья каждые 1000 часов
        IF (VIO_Health_Data.Total_Runtime_Hours MOD 1000) = 0 THEN
            VIO_Health_Data.Health_Score := TO_BYTE(LIMIT(0, TO_INT(VIO_Health_Data.Health_Score) - 1, 100));
        END_IF;
        
        // Анализ рабочего тока (после пускового режима)
        IF (VI_System_Time_MS - L_Start_Time) > 10000 THEN // 10 секунд после пуска
            IF VI_Current_Value > (VI_Nominal_Value * 1.1) THEN
                // Повышенный рабочий ток - ускоренный износ (-1% в час)
                VIO_Health_Data.Health_Score := TO_BYTE(LIMIT(0, TO_INT(VIO_Health_Data.Health_Score) - 1, 100));
            END_IF;
        END_IF;
    END_IF;
END_IF;

// 4. Генерация предупреждения
IF VIO_Health_Data.Health_Score < 20 THEN
    VIO_Health_Data.Maintenance_Required := TRUE;
    VIO_Health_Data.Warning_Message := 'Критический износ: проверьте механику';
ELSIF VIO_Health_Data.Health_Score < 60 THEN
    VIO_Health_Data.Maintenance_Required := FALSE;
    VIO_Health_Data.Warning_Message := 'Предупреждение: повышенное трение';
ELSE
    VIO_Health_Data.Maintenance_Required := FALSE;
    VIO_Health_Data.Warning_Message := 'В норме';
END_IF;

L_Prev_Running := VI_Is_Running;
          
END_FUNCTION_BLOCK

FUNCTION_BLOCK FB_Analog_Validator
  VAR_INPUT
    VI_Value : REAL;
    VI_Min_Valid : REAL;
    VI_Max_Valid : REAL;
    VI_Fallback_Mode : INT := 0;
    VI_Default_Value : REAL := 0.0;
  END_VAR
  VAR_OUTPUT
    VO_Value : REAL;
    VO_Error : BOOL;
  END_VAR
  VAR
    L_Last_Good_Value : REAL;
    L_First_Valid : BOOL := FALSE;
  END_VAR

            IF VI_Value >= VI_Min_Valid AND VI_Value <= VI_Max_Valid THEN
    VO_Error := FALSE;
    VO_Value := VI_Value;
    L_Last_Good_Value := VI_Value;
    L_First_Valid := TRUE;
ELSE
    VO_Error := TRUE;
    IF VI_Fallback_Mode = 1 OR NOT L_First_Valid THEN
        VO_Value := VI_Default_Value;
    ELSE
        VO_Value := L_Last_Good_Value;
    END_IF;
END_IF;
// >>> BULK_SYNC_ANCHOR: FB_Analog_Validator <<<
          
END_FUNCTION_BLOCK

FUNCTION_BLOCK FB_FloorHeating_Controller
  VAR_INPUT
    VI_Current_Temp : REAL;
    VI_Config : ST_FloorHeating_Circuit_Config;
    VI_Tariff : ST_Tariff_Config;
    VI_Current_Hour : UINT;
    VI_IsActivePLC : BOOL;
    VI_System_Time_MS : UDINT;
  END_VAR
  VAR_OUTPUT
    VO_Pump_Run : BOOL;
    VO_Valve_Pos : REAL;
    VO_Valve_Bool : BOOL;
    VO_Effective_Setpoint : REAL;
  END_VAR
  VAR
    L_Is_Night : BOOL;
    L_PID : FB_PID_Controller;
    L_Last_Time : UDINT;
    L_Cycle_Time_S : REAL;
    L_PWM_Period_MS : UDINT;
    L_PWM_Duty_MS : UDINT;
    L_Current_Phase_MS : UDINT;
    L_PWM_Start_Time : UDINT;
  END_VAR

            // Вычисление времени цикла
IF L_Last_Time = 0 THEN
    L_Last_Time := VI_System_Time_MS;
    L_Cycle_Time_S := 1.0;
ELSE
    L_Cycle_Time_S := UDINT_TO_REAL((SEL(VI_System_Time_MS >= L_Last_Time, VI_System_Time_MS - L_Last_Time, (4294967295 - L_Last_Time) + VI_System_Time_MS + 1))) / 1000.0;
    L_Last_Time := VI_System_Time_MS;
END_IF;
IF L_Cycle_Time_S <= 0.0 THEN L_Cycle_Time_S := 0.01; END_IF;

// 1. Определение активного тарифа
IF VI_Tariff.Enabled THEN
    IF VI_Tariff.Night_Start_Hour > VI_Tariff.Night_End_Hour THEN
        // Переход через полночь (например, 23:00 - 07:00)
        L_Is_Night := (VI_Current_Hour >= VI_Tariff.Night_Start_Hour) OR (VI_Current_Hour < VI_Tariff.Night_End_Hour);
    ELSE
        // В пределах одного дня
        L_Is_Night := (VI_Current_Hour >= VI_Tariff.Night_Start_Hour) AND (VI_Current_Hour < VI_Tariff.Night_End_Hour);
    END_IF;
ELSE
    L_Is_Night := FALSE;
END_IF;

// 2. Расчет эффективной уставки
VO_Effective_Setpoint := VI_Config.design_temp;
IF L_Is_Night THEN
    VO_Effective_Setpoint := VO_Effective_Setpoint + VI_Tariff.Boost_Delta;
END_IF;

// 3. ПИД-регулирование
L_PID(
    VI_SetPoint := VO_Effective_Setpoint,
    VI_ProcessValue := VI_Current_Temp,
    VI_Kp := VI_Config.pid_kp,
    VI_Tn := 300.0,
    VI_Tv := 0.0,
    VI_Y_Min := 0.0,
    VI_Y_Max := 100.0,
    VI_Cycle_Time_S := L_Cycle_Time_S,
    VO_Output => VO_Valve_Pos
);

// 4. ШИМ-модуляция для термоэлектрического привода
IF VI_Config.pwm_period_s > 0 THEN
    L_PWM_Period_MS := TO_UDINT(VI_Config.pwm_period_s) * 1000;
ELSE
    L_PWM_Period_MS := 600000; // 10 минут
END_IF;

L_Current_Phase_MS := (SEL(VI_System_Time_MS >= L_PWM_Start_Time, VI_System_Time_MS - L_PWM_Start_Time, (4294967295 - L_PWM_Start_Time) + VI_System_Time_MS + 1));
IF L_Current_Phase_MS >= L_PWM_Period_MS THEN
    L_PWM_Start_Time := VI_System_Time_MS - (L_Current_Phase_MS - L_PWM_Period_MS); // Сохраняем остаток для точности
    L_Current_Phase_MS := (SEL(VI_System_Time_MS >= L_PWM_Start_Time, VI_System_Time_MS - L_PWM_Start_Time, (4294967295 - L_PWM_Start_Time) + VI_System_Time_MS + 1));
END_IF;

L_PWM_Duty_MS := TO_UDINT((VO_Valve_Pos / 100.0) * TO_REAL(L_PWM_Period_MS));

IF VI_IsActivePLC THEN
    VO_Pump_Run := (VO_Valve_Pos > 5.0);
    
    IF VO_Valve_Pos >= 100.0 THEN
        VO_Valve_Bool := TRUE;
    ELSIF VO_Valve_Pos <= 0.0 THEN
        VO_Valve_Bool := FALSE;
    ELSE
        VO_Valve_Bool := (L_Current_Phase_MS <= L_PWM_Duty_MS);
    END_IF;
ELSE
    VO_Pump_Run := FALSE;
    VO_Valve_Bool := FALSE;
END_IF;
          
END_FUNCTION_BLOCK

FUNCTION_BLOCK FB_Heating_Boiler_Control
  VAR_INPUT
    VI_System_Time_MS : UDINT;
    VI_IsActivePLC : BOOL;
    VI_DHW_Heating_Demand : BOOL;
    VI_DHW_Target_Temp : REAL;
    VI_Target_Supply_Temp : REAL;
    VI_Freeze_Mode_Active : BOOL;
    VI_Policy_Degraded : BOOL;
    VI_Manifold_Pumps : ARRAY[1..GVL_CONSTANTS.C_MAX_MANIFOLDS] OF BOOL;
    VI_Manifold_Valves : ARRAY[1..GVL_CONSTANTS.C_MAX_MANIFOLDS] OF REAL;
    VI_Boiler_Flame_Status : ARRAY[1..GVL_CONSTANTS.C_MAX_BOILERS] OF BOOL;
    VI_Boiler_Error_Status : ARRAY[1..GVL_CONSTANTS.C_MAX_BOILERS] OF BOOL;
    VI_Boiler_OT_Online : ARRAY[1..GVL_CONSTANTS.C_MAX_BOILERS] OF BOOL;
  END_VAR
  VAR_OUTPUT
    VO_Boiler_OT_Enable : ARRAY[1..GVL_CONSTANTS.C_MAX_BOILERS] OF BOOL;
    VO_Boiler_OT_Setpoint : ARRAY[1..GVL_CONSTANTS.C_MAX_BOILERS] OF REAL;
    VO_Boiler_Status : ARRAY[1..GVL_CONSTANTS.C_MAX_BOILERS] OF ST_Boiler_Status;
    VO_Any_Subsystem_Degraded : BOOL;
    VO_Lead_Boiler : BYTE;
    VO_Demand_Power : REAL;
  END_VAR
  VAR_IN_OUT
    VI_Boiler_Modulation : ARRAY[1..GVL_CONSTANTS.C_MAX_BOILERS] OF REAL;
  END_VAR
  VAR
    L_i : INT;
    L_Delta_MS : UDINT;
    L_Last_Scan_Time : UDINT;
    L_Scan_Time_Init : BOOL := FALSE;
    L_Boiler_Request_Enable : ARRAY[1..GVL_CONSTANTS.C_MAX_BOILERS] OF BOOL;
    L_Boiler_Request_Setpoint : ARRAY[1..GVL_CONSTANTS.C_MAX_BOILERS] OF REAL;
    L_Boiler_OT_Command_Valid : ARRAY[1..GVL_CONSTANTS.C_MAX_BOILERS] OF BOOL;
    L_Boiler_Life : ARRAY[1..GVL_CONSTANTS.C_MAX_BOILERS] OF FB_Lifetime_Predictor;
    fbBoilerCascade : FB_Boiler_Cascade_Manager;
    fbBoilerOpenTherm : FB_Boiler_OpenTherm_Interface;
  END_VAR

            // ==============================================================================
// Heating boiler control helper
//
// Internal refactoring helper for FB_Heating_System_Manager.
// Owns demand aggregation, boiler cascade request, OpenTherm transport,
// status normalization, degradation projection, and boiler resource accounting.
// ==============================================================================



VO_Any_Subsystem_Degraded := FALSE;
VO_Demand_Power := 0.0;

FOR L_i := 1 TO GVL_CONSTANTS.C_MAX_MANIFOLDS DO
    IF VI_Manifold_Pumps[L_i] THEN
        VO_Demand_Power := VO_Demand_Power + VI_Manifold_Valves[L_i];
    END_IF;
END_FOR;

IF VI_Freeze_Mode_Active AND VO_Demand_Power < 20.0 THEN
    VO_Demand_Power := 20.0;
END_IF;

IF VI_Policy_Degraded THEN
    IF VO_Demand_Power > 60.0 THEN
        VO_Demand_Power := 60.0;
    END_IF;
END_IF;

fbBoilerCascade(
    VI_Enable := VI_IsActivePLC AND ((VO_Demand_Power > GVL_CONSTANTS.C_BOILER_CASCADE_MIN_DEMAND) OR VI_Freeze_Mode_Active),
    VI_System_Time_MS := VI_System_Time_MS,
    VI_Boiler_Stop := FALSE,
    VI_DHW_Heating_Demand := VI_DHW_Heating_Demand,
    VI_DHW_Target_Temp := VI_DHW_Target_Temp,
    VI_Target_Supply_Temp := VI_Target_Supply_Temp,
    VI_Demand_Power := VO_Demand_Power,
    VI_Boiler_Flame_Status := VI_Boiler_Flame_Status,
    VI_Boiler_Error_Status := VI_Boiler_Error_Status,
    VI_Boiler_OT_Online := VI_Boiler_OT_Online,
    VI_Boiler_Modulation := VI_Boiler_Modulation,
    VO_Boiler_Enable => L_Boiler_Request_Enable,
    VO_Boiler_Setpoint => L_Boiler_Request_Setpoint,
    VO_Lead_Boiler => VO_Lead_Boiler
);

FOR L_i := 1 TO GVL_CONSTANTS.C_MAX_BOILERS DO
    IF NOT VI_Boiler_OT_Online[L_i] OR VI_Boiler_Error_Status[L_i] THEN
        L_Boiler_Request_Enable[L_i] := FALSE;
        L_Boiler_Request_Setpoint[L_i] := 0.0;
    END_IF;
END_FOR;

fbBoilerOpenTherm(
    VI_Enable := L_Boiler_Request_Enable,
    VI_Setpoint := L_Boiler_Request_Setpoint,
    VI_OT_Online := VI_Boiler_OT_Online,
    VI_OT_Error := VI_Boiler_Error_Status,
    VO_OT_Enable => VO_Boiler_OT_Enable,
    VO_OT_Setpoint => VO_Boiler_OT_Setpoint,
    VO_OT_Command_Valid => L_Boiler_OT_Command_Valid
);

FOR L_i := 1 TO GVL_CONSTANTS.C_MAX_BOILERS DO
    VO_Boiler_Status[L_i].Active := L_Boiler_Request_Enable[L_i];
    VO_Boiler_Status[L_i].Warning := FALSE;
    VO_Boiler_Status[L_i].Error := FALSE;

    IF NOT VI_Boiler_OT_Online[L_i] THEN
        VO_Boiler_Status[L_i].Error := TRUE;
        VO_Boiler_Status[L_i].Error_ID := TO_WORD(GVL_CONFIG.ERR_BOILER_OFFLINE);
        VO_Any_Subsystem_Degraded := TRUE;
    ELSIF VI_Boiler_Error_Status[L_i] THEN
        VO_Boiler_Status[L_i].Error := TRUE;
        VO_Boiler_Status[L_i].Error_ID := TO_WORD(GVL_CONFIG.ERR_BOILER_GENERAL_FAULT);
        VO_Any_Subsystem_Degraded := TRUE;
    ELSIF L_Boiler_Request_Enable[L_i] AND NOT VI_Boiler_Flame_Status[L_i] THEN
        VO_Boiler_Status[L_i].Warning := TRUE;
        VO_Boiler_Status[L_i].Error_ID := TO_WORD(GVL_CONFIG.ERR_BOILER_NO_FLAME);
        VO_Any_Subsystem_Degraded := TRUE;
    ELSE
        VO_Boiler_Status[L_i].Error_ID := 0;
    END_IF;
END_FOR;

IF NOT L_Scan_Time_Init THEN
    L_Last_Scan_Time := VI_System_Time_MS;
    L_Scan_Time_Init := TRUE;
END_IF;

L_Delta_MS := (SEL(VI_System_Time_MS >= L_Last_Scan_Time, VI_System_Time_MS - L_Last_Scan_Time, (4294967295 - L_Last_Scan_Time) + VI_System_Time_MS + 1));
IF L_Delta_MS > 1000 THEN
    L_Delta_MS := 1000;
END_IF;

L_Last_Scan_Time := VI_System_Time_MS;

FOR L_i := 1 TO GVL_CONSTANTS.C_MAX_BOILERS DO
    VO_Boiler_Status[L_i].Work_Seconds := GVL_Retain.G_Boiler_Work_Seconds[L_i];

    IF VI_Boiler_Flame_Status[L_i] THEN
        GVL_Retain.G_Boiler_Accumulated_MS[L_i] := GVL_Retain.G_Boiler_Accumulated_MS[L_i] + L_Delta_MS;
        IF GVL_Retain.G_Boiler_Accumulated_MS[L_i] >= GVL_CONSTANTS.C_MS_IN_SECOND THEN
            GVL_Retain.G_Boiler_Work_Seconds[L_i] := GVL_Retain.G_Boiler_Work_Seconds[L_i] + (GVL_Retain.G_Boiler_Accumulated_MS[L_i] / 1000);
            GVL_Retain.G_Boiler_Accumulated_MS[L_i] := GVL_Retain.G_Boiler_Accumulated_MS[L_i] MOD 1000;

            IF GVL_Retain.G_Boiler_Work_Seconds[L_i] > 4000000000 THEN
                GVL_Retain.G_Boiler_Work_Seconds[L_i] := 0;
            END_IF;

            VO_Boiler_Status[L_i].Work_Seconds := GVL_Retain.G_Boiler_Work_Seconds[L_i];
        END_IF;
    END_IF;

    VO_Boiler_Status[L_i].Work_Hours := TO_REAL(VO_Boiler_Status[L_i].Work_Seconds) / 3600.0;

    L_Boiler_Life[L_i](
        VI_Runtime_Hours := TO_UDINT(VO_Boiler_Status[L_i].Work_Hours),
        VI_Start_Count := 0,
        VI_Nominal_Life := 50000
    );
    VO_Boiler_Status[L_i].Resource_Percent := TO_REAL(L_Boiler_Life[L_i].VO_Remaining_Percent);
    VO_Boiler_Status[L_i].Running := VI_Boiler_Flame_Status[L_i];
END_FOR;

// >>> BULK_SYNC_ANCHOR: FB_Heating_Boiler_Control <<<
          
END_FUNCTION_BLOCK

FUNCTION_BLOCK FB_Watchdog
  VAR_INPUT
    VI_System_Time_MS : UDINT;
    VI_Timeout_MS : UDINT := 2000;
  END_VAR
  VAR_OUTPUT
    VO_Alive : BOOL;
    VO_Watchdog_Fault : BOOL;
    VO_Cycle_DT_MS : UDINT;
  END_VAR
  VAR
    L_Initialized : BOOL := FALSE;
    L_Last_Call_MS : UDINT := 0;
    L_DT_MS : UDINT := 0;
  END_VAR

            IF NOT L_Initialized THEN
    L_Initialized := TRUE;
    L_Last_Call_MS := VI_System_Time_MS;
    VO_Cycle_DT_MS := 0;
    VO_Watchdog_Fault := FALSE;
    VO_Alive := TRUE;
    RETURN;
END_IF;

// Measure real time gap between successive calls
L_DT_MS := (SEL(VI_System_Time_MS >= L_Last_Call_MS, VI_System_Time_MS - L_Last_Call_MS, (4294967295 - L_Last_Call_MS) + VI_System_Time_MS + 1));
VO_Cycle_DT_MS := L_DT_MS;

// Fault if the task/cycle resumed after an abnormal pause
VO_Watchdog_Fault := (L_DT_MS > VI_Timeout_MS);
VO_Alive := NOT VO_Watchdog_Fault;

// Store current timestamp for next cycle
L_Last_Call_MS := VI_System_Time_MS;
// >>> BULK_SYNC_ANCHOR: FB_Watchdog <<<
          
END_FUNCTION_BLOCK

FUNCTION_BLOCK FB_DHW_Manager
  VAR_INPUT
    VI_System_Time_MS : UDINT;
    VI_Current_TOD : TOD;
    VI_IsActivePLC : BOOL;
    VI_Temp : REAL;
    VI_Pressure : REAL;
    VI_Config : ST_DHW_Config;
    VI_Current_Day_Of_Week : UINT;
    VI_Reset_Errors : BOOL;
    VI_Emergency_Stop : BOOL;
    VI_System_Mode : E_System_Operating_Mode;
    VI_IO_Modules_Online : ARRAY[1..GVL_CONSTANTS.C_MAX_MODULES] OF BOOL;
  END_VAR
  VAR_OUTPUT
    VO_Status : ST_DHW_Status;
    VO_Heating_Pump : BOOL;
    VO_Circ_Pump : BOOL;
  END_VAR
  VAR
    L_i : INT;
    L_Current_TOD : TOD;
    L_Legionella_Active : BOOL;
    L_Legionella_Timer : FB_System_Timer;
    L_Last_Good_Temp : REAL := 55.0;
    L_Legionella_Done_Today : BOOL;
    L_Last_Legionella_Day : UINT;
    fbTempValidator : FB_Analog_Validator;
    fbPressValidator : FB_Analog_Validator;
    L_Error_Latched : BOOL;
    L_Error_ID_Latched : WORD;
    L_Policy_Degraded : BOOL;
    L_Policy_Freeze_Protection : BOOL;
    L_Policy_Safe_Stop : BOOL;
    L_Target_Temp_Adjusted : REAL;
  END_VAR

            // >>> SYNC_TEST_MARKER_001 <<<


IF NOT VI_IsActivePLC THEN RETURN; END_IF;


GVL_STATE.G_DHW_IO_Fault := FALSE;
GVL_STATE.G_DHW_Sensor_Fault := FALSE;
GVL_STATE.G_DHW_Subsystem_Degraded := FALSE;

IF VI_Emergency_Stop THEN
    VO_Heating_Pump := FALSE;
    VO_Circ_Pump := FALSE;
    VO_Status.Warning := FALSE;
    VO_Status.Error := TRUE;
    VO_Status.Error_ID := TO_WORD(GVL_CONFIG.ERR_DHW_IO_OFFLINE); // временно используем общий аварийный код до детализации safety-кодов
    VO_Status.Heating_Pump_On := FALSE;
    VO_Status.Circ_Pump_On := FALSE;
    RETURN;
END_IF;

// Фиксация текущего времени
L_Current_TOD := VI_Current_TOD;

// ========================================
// DHW POLICY LAYER
// ========================================
L_Policy_Safe_Stop := (VI_System_Mode = E_System_Operating_Mode.MODE_SAFE_STOP);
L_Policy_Freeze_Protection := (VI_System_Mode = E_System_Operating_Mode.MODE_FREEZE_PROTECTION);
L_Policy_Degraded := (VI_System_Mode = E_System_Operating_Mode.MODE_DEGRADED);
L_Target_Temp_Adjusted := VI_Config.Target_Temp;
IF L_Policy_Degraded THEN
    L_Target_Temp_Adjusted := VI_Config.Target_Temp - VI_Config.Degraded_Target_Delta;
END_IF;

// ========================================
// DHW POLICY OVERRIDE
// ========================================
IF L_Policy_Safe_Stop THEN
    VO_Heating_Pump := FALSE;
    VO_Circ_Pump := FALSE;
    RETURN;
END_IF;

IF L_Policy_Freeze_Protection THEN
    VO_Heating_Pump := FALSE;
    VO_Circ_Pump := FALSE;
    RETURN;
END_IF;

// Сброс признака выполнения термодезинфекции при смене дня.
IF L_Last_Legionella_Day <> VI_Current_Day_Of_Week THEN
    L_Legionella_Done_Today := FALSE;
    L_Last_Legionella_Day := VI_Current_Day_Of_Week;
END_IF;

// Базовый сброс незащёлкнутых статусных флагов на текущий цикл.
// Критические ошибки ниже могут зафиксироваться и завершить выполнение через RETURN.
VO_Status.Warning := FALSE;
VO_Status.Error := FALSE;
VO_Status.Error_ID := 0;

// Сброс ошибок
IF VI_Reset_Errors THEN
    L_Error_Latched := FALSE;
    L_Error_ID_Latched := 0;
END_IF;

// Проверка связи с модулями ввода-вывода
FOR L_i := 1 TO GVL_CONSTANTS.C_MAX_MODULES DO
    IF NOT VI_IO_Modules_Online[L_i] THEN
        L_Error_Latched := TRUE;
        GVL_STATE.G_DHW_IO_Fault := TRUE;
        L_Error_ID_Latched := TO_WORD(GVL_CONFIG.ERR_DHW_IO_OFFLINE); // Потеря связи с модулями ввода-вывода
    END_IF;
END_FOR;

// 1. Обработка неисправностей датчиков и сервисных режимов (ТЗ 7.0)
fbTempValidator(
    VI_Value := VI_Temp,
    VI_Min_Valid := 0.0,
    VI_Max_Valid := 100.0,
    VI_Fallback_Mode := 0,
    VI_Default_Value := 55.0
);

fbPressValidator(
    VI_Value := VI_Pressure,
    VI_Min_Valid := 0.0,
    VI_Max_Valid := 10.0,
    VI_Fallback_Mode := 0
);

VO_Status.Temp := fbTempValidator.VO_Value;
VO_Status.Pressure := fbPressValidator.VO_Value;

// Сохраняем последнее достоверное значение температуры ГВС.
// Используется только для диагностики/сервиса, не для fallback-управления.
IF NOT fbTempValidator.VO_Error THEN
    L_Last_Good_Temp := VO_Status.Temp;
END_IF;

IF fbTempValidator.VO_Error THEN
    GVL_STATE.G_DHW_Sensor_Fault := TRUE;
    L_Error_Latched := TRUE;
    L_Error_ID_Latched := TO_WORD(GVL_CONFIG.ERR_DHW_TEMP_SENSOR_FAULT); // Критическая ошибка датчика температуры
ELSIF (VO_Status.Pressure < 1.0 OR VO_Status.Pressure > 4.0) AND NOT fbPressValidator.VO_Error THEN
    L_Error_Latched := TRUE;
    L_Error_ID_Latched := TO_WORD(GVL_CONFIG.ERR_DHW_PRESSURE_OUT_OF_RANGE); // Давление вне нормы
END_IF;

IF L_Error_Latched THEN
    // Критическая ошибка: переход в безопасное состояние с полной остановкой насосов.
    VO_Heating_Pump := FALSE;
    VO_Circ_Pump := FALSE;
    VO_Status.Warning := FALSE;
    VO_Status.Error := TRUE;
    VO_Status.Error_ID := L_Error_ID_Latched;
    VO_Status.Heating_Pump_On := FALSE;
    VO_Status.Circ_Pump_On := FALSE;
    RETURN;
END_IF;

// Ошибка датчика давления не останавливает ГВС,
// но переводит подсистему в режим предупреждения (degraded mode).
IF fbPressValidator.VO_Error THEN
    GVL_STATE.G_DHW_Sensor_Fault := TRUE;
    GVL_STATE.G_DHW_Subsystem_Degraded := TRUE;
    VO_Status.Warning := TRUE;
    VO_Status.Error := FALSE;
    VO_Status.Error_ID := TO_WORD(GVL_CONFIG.ERR_DHW_PRESSURE_SENSOR_FAULT);
END_IF;

// 2. Логика поддержания температуры воды в бойлере (Нагрев)
// На этом этапе FB уже выполняется только на активном ПЛК.
    
// Термическая дезинфекция (Легионелла)
IF VI_Config.Anti_Legionella_Enabled
   AND (VI_Current_Day_Of_Week = VI_Config.Anti_Legionella_Day)
   AND (L_Current_TOD >= TOD#02:00)
   AND (L_Current_TOD <= TOD#04:00)
   AND NOT L_Legionella_Done_Today THEN
    L_Legionella_Active := TRUE;
ELSE
    L_Legionella_Active := FALSE;
END_IF;

L_Legionella_Timer(IN := L_Legionella_Active AND VO_Status.Temp >= 70.0, PT := T#30m, VI_System_Time_MS := VI_System_Time_MS);
IF L_Legionella_Timer.Q THEN
    L_Legionella_Active := FALSE; // Дезинфекция завершена
    L_Legionella_Done_Today := TRUE; // Повторно в те же сутки не запускать
END_IF;

// Двухпозиционное регулирование с гистерезисом
IF L_Legionella_Active THEN
    IF VO_Status.Temp < 70.0 THEN
        VO_Heating_Pump := TRUE;
    ELSIF VO_Status.Temp > 72.0 THEN
        VO_Heating_Pump := FALSE;
    END_IF;
ELSE
    IF VO_Status.Temp < (L_Target_Temp_Adjusted - VI_Config.Hysteresis) THEN
        VO_Heating_Pump := TRUE;
    ELSIF VO_Status.Temp > (L_Target_Temp_Adjusted + VI_Config.Hysteresis) THEN
        VO_Heating_Pump := FALSE;
    END_IF;
END_IF;

// 3. Управление циркуляционным насосом ГВС по расписанию
// Рециркуляция обеспечивает мгновенное наличие горячей воды у потребителя
VO_Circ_Pump := SEL(VI_Config.Circulation_Schedule_Enabled AND NOT (VI_Config.Night_Mode_Enabled AND (L_Current_TOD < VI_Config.Circulation_Start OR L_Current_TOD > VI_Config.Circulation_End)), FALSE, TRUE);

// Формирование статусных данных для визуализации.
// К этому моменту статус уже консистентен:
// - Error = критическая ошибка с остановкой ГВС
// - Warning = деградация без остановки
VO_Status.Heating_Pump_On := VO_Heating_Pump;
VO_Status.Circ_Pump_On := VO_Circ_Pump;

// >>> BULK_SYNC_ANCHOR: FB_DHW_Manager <<<
          
END_FUNCTION_BLOCK

FUNCTION_BLOCK FB_System_Intent_Publisher
  VAR_INPUT
    VI_System_Time_MS : UDINT;
    VI_Gateway_Writes_Allowed : BOOL;
  END_VAR

            // ==============================================================================
// System intent publisher helper
//
// Internal helper for PRG_System.
// Owns publication of system-mode gates into GVL_INTENT_SYSTEM.
// ==============================================================================



GVL_INTENT_SYSTEM.I_Source_Valid := TRUE;
GVL_INTENT_SYSTEM.I_Last_Update_MS := VI_System_Time_MS;
GVL_INTENT_SYSTEM.I_Mode_Safe_Stop_Active := (GVL_STATE.G_System_Mode = E_System_Operating_Mode.MODE_SAFE_STOP);
GVL_INTENT_SYSTEM.I_Mode_Degraded_Active := (GVL_STATE.G_System_Mode = E_System_Operating_Mode.MODE_DEGRADED);
GVL_INTENT_SYSTEM.I_Mode_Freeze_Protection_Active := (GVL_STATE.G_System_Mode = E_System_Operating_Mode.MODE_FREEZE_PROTECTION);
GVL_INTENT_SYSTEM.I_Operator_Scenario_Block := (GVL_STATE.G_System_Mode = E_System_Operating_Mode.MODE_SAFE_STOP);
GVL_INTENT_SYSTEM.I_Lighting_Overrides_Block := (GVL_STATE.G_System_Mode = E_System_Operating_Mode.MODE_SAFE_STOP);
GVL_INTENT_SYSTEM.I_Blinds_Overrides_Block := (GVL_STATE.G_System_Mode = E_System_Operating_Mode.MODE_SAFE_STOP);
GVL_INTENT_SYSTEM.I_Socket_Overrides_Block := (GVL_STATE.G_System_Mode = E_System_Operating_Mode.MODE_SAFE_STOP);
GVL_INTENT_SYSTEM.I_Gateway_Writes_Allowed := VI_Gateway_Writes_Allowed;
GVL_INTENT_SYSTEM.I_Scenario_Request_Allowed := (GVL_STATE.G_System_Mode <> E_System_Operating_Mode.MODE_SAFE_STOP);

// >>> BULK_SYNC_ANCHOR: FB_System_Intent_Publisher <<<
          
END_FUNCTION_BLOCK

FUNCTION_BLOCK FB_Heating_Decision_Context
  VAR_INPUT
    VI_Manifold_Pump_In_Service : ARRAY[1..GVL_CONSTANTS.C_MAX_MANIFOLDS] OF BOOL;
    VI_Manifold_Pressure_Fault : ARRAY[1..GVL_CONSTANTS.C_MAX_MANIFOLDS] OF BOOL;
    VI_Manifold_Current_Fault : ARRAY[1..GVL_CONSTANTS.C_MAX_MANIFOLDS] OF BOOL;
    VI_Manifold_Thermal_Weight : ARRAY[1..GVL_CONSTANTS.C_MAX_MANIFOLDS] OF REAL;
    VI_Manifold_Priority : ARRAY[1..GVL_CONSTANTS.C_MAX_MANIFOLDS] OF INT;
    VI_Max_Thermal_Budget : REAL;
  END_VAR
  VAR_OUTPUT
    VO_Manifold_Allowed : ARRAY[1..GVL_CONSTANTS.C_MAX_MANIFOLDS] OF BOOL;
    VO_Manifold_Enabled : ARRAY[1..GVL_CONSTANTS.C_MAX_MANIFOLDS] OF BOOL;
    VO_Heating_Degraded : BOOL;
  END_VAR
  VAR
    L_i : INT;
    L_j : INT;
    L_Used : REAL;
    L_Selected : ARRAY[1..GVL_CONSTANTS.C_MAX_MANIFOLDS] OF BOOL;
    L_MaxPriority : INT;
    L_CurrentPriority : INT;
  END_VAR

            VO_Heating_Degraded := FALSE;

// STEP 1: Allowed
FOR L_i := 1 TO GVL_CONSTANTS.C_MAX_MANIFOLDS DO
    VO_Manifold_Allowed[L_i] := TRUE;

    IF NOT VI_Manifold_Pump_In_Service[L_i] THEN
        VO_Manifold_Allowed[L_i] := FALSE;
    END_IF;

    IF VI_Manifold_Pressure_Fault[L_i] THEN
        VO_Manifold_Allowed[L_i] := FALSE;
    END_IF;

    IF VI_Manifold_Current_Fault[L_i] THEN
        VO_Manifold_Allowed[L_i] := FALSE;
    END_IF;

    IF NOT VO_Manifold_Allowed[L_i] THEN
        VO_Heating_Degraded := TRUE;
    END_IF;
END_FOR;

// STEP 2: find max priority
L_MaxPriority := 0;
FOR L_i := 1 TO GVL_CONSTANTS.C_MAX_MANIFOLDS DO
    IF VI_Manifold_Priority[L_i] > L_MaxPriority THEN
        L_MaxPriority := VI_Manifold_Priority[L_i];
    END_IF;
END_FOR;

// STEP 3: allocation by priority + budget
FOR L_i := 1 TO GVL_CONSTANTS.C_MAX_MANIFOLDS DO
    VO_Manifold_Enabled[L_i] := FALSE;
END_FOR;

L_Used := 0.0;

FOR L_CurrentPriority := L_MaxPriority TO 1 BY -1 DO

    FOR L_i := 1 TO GVL_CONSTANTS.C_MAX_MANIFOLDS DO

        IF (VI_Manifold_Priority[L_i] = L_CurrentPriority) AND VO_Manifold_Allowed[L_i] THEN

            IF (L_Used + VI_Manifold_Thermal_Weight[L_i]) <= VI_Max_Thermal_Budget THEN
                VO_Manifold_Enabled[L_i] := TRUE;
                L_Used := L_Used + VI_Manifold_Thermal_Weight[L_i];
            END_IF;

        END_IF;

    END_FOR;

END_FOR;
          
END_FUNCTION_BLOCK

FUNCTION_BLOCK FB_State_Snapshot_Manager
  VAR_INPUT
    VI_System_Time_MS : UDINT;
    VI_Trigger_Event : BOOL;
    VI_Event_Code : WORD;
    VI_Current_State : ST_State_Snapshot;
  END_VAR
  VAR_OUTPUT
    VO_Snapshot_Saved : BOOL;
  END_VAR
  VAR
    L_Snapshot_Buffer : ARRAY[1..GVL_CONSTANTS.C_MAX_STATE_SNAPSHOTS] OF ST_State_Snapshot;
    L_Write_Idx : INT := 1;
  END_VAR

            IF VI_Trigger_Event THEN
    L_Snapshot_Buffer[L_Write_Idx] := VI_Current_State;
    L_Snapshot_Buffer[L_Write_Idx].timestamp_ms := VI_System_Time_MS;
    
    // NOTE:
    // ST_State_Snapshot no longer contains trigger_event_code in live project.
    // VI_Event_Code is reserved for future snapshot metadata extension.
    
    L_Write_Idx := (L_Write_Idx MOD GVL_CONSTANTS.C_MAX_STATE_SNAPSHOTS) + 1;
    VO_Snapshot_Saved := TRUE;
ELSE
    VO_Snapshot_Saved := FALSE;
END_IF;
          
END_FUNCTION_BLOCK

FUNCTION_BLOCK FB_Lifetime_Manager
  VAR_INPUT
    VI_System_Time_MS : UDINT;
    VI_Device_Active : BOOL;
    VI_Device_ID : BYTE;
    VI_Nominal_Hours : UDINT;
  END_VAR
  VAR_IN_OUT
    VIO_Status : ST_Lifetime_Status;
  END_VAR
  VAR
    L_Last_Time : UDINT;
    L_Prev_State : BOOL;
    L_Delta_MS : UDINT;
    L_Runtime_Accum_MS : UDINT;
    L_Remaining_Percent_UDINT : UDINT;
  END_VAR

            // === DELTA TIME ===
IF VI_System_Time_MS >= L_Last_Time THEN
    L_Delta_MS := VI_System_Time_MS - L_Last_Time;
ELSE
    // overflow
    L_Delta_MS := (4294967295 - L_Last_Time) + VI_System_Time_MS + 1;
END_IF;

L_Last_Time := VI_System_Time_MS;

// === START COUNT ===
IF VI_Device_Active AND NOT L_Prev_State THEN
    VIO_Status.start_count := VIO_Status.start_count + 1;
END_IF;

L_Prev_State := VI_Device_Active;

// === RUNTIME ACCUMULATION ===
IF VI_Device_Active THEN
    L_Runtime_Accum_MS := L_Runtime_Accum_MS + L_Delta_MS;

    WHILE L_Runtime_Accum_MS >= 3600000 DO
        VIO_Status.runtime_hours := VIO_Status.runtime_hours + 1;
        L_Runtime_Accum_MS := L_Runtime_Accum_MS - 3600000;
    END_WHILE;
END_IF;

// === BASIC LIFETIME ESTIMATION ===
IF VI_Nominal_Hours > 0 THEN
    IF VIO_Status.runtime_hours >= VI_Nominal_Hours THEN
        VIO_Status.remaining_hours := 0;
        VIO_Status.remaining_percent := 0;
    ELSE
        VIO_Status.remaining_hours := VI_Nominal_Hours - VIO_Status.runtime_hours;
        L_Remaining_Percent_UDINT := (VIO_Status.remaining_hours * 100) / VI_Nominal_Hours;

        IF L_Remaining_Percent_UDINT > 100 THEN
            L_Remaining_Percent_UDINT := 100;
        END_IF;

        VIO_Status.remaining_percent := UDINT_TO_BYTE(L_Remaining_Percent_UDINT);
    END_IF;
ELSE
    VIO_Status.remaining_hours := 0;
    VIO_Status.remaining_percent := 0;
END_IF;

VIO_Status.maintenance_required := VIO_Status.remaining_percent <= GVL_Lifetime.G_Maintenance_Threshold_Percent;

// === BASIC FLAGS ===
VIO_Status.device_id := VI_Device_ID;
VIO_Status.last_calc_timestamp := VI_System_Time_MS;
          
END_FUNCTION_BLOCK

FUNCTION_BLOCK FB_SHA1
  VAR_INPUT
    Length : INT;
  END_VAR
  VAR_OUTPUT
    Hash : ARRAY[0..19] OF BYTE;
  END_VAR
  VAR_IN_OUT
    Data : ARRAY[0..127] OF BYTE;
  END_VAR
  VAR
    H0, H1, H2, H3, H4 : DWORD;
    A, B, C, D, E, F, K, Temp : DWORD;
    W : ARRAY[0..79] OF DWORD;
    i, j, t : INT;
    PaddedData : ARRAY[0..127] OF BYTE;
    PaddedLength : INT;
    NumBlocks : INT;
    BlockOffset : INT;
  END_VAR

            // Initialize variables
H0 := 16#67452301;
H1 := 16#EFCDAB89;
H2 := 16#98BADCFE;
H3 := 16#10325476;
H4 := 16#C3D2E1F0;

// Pre-processing
FOR i := 0 TO Length - 1 DO
    PaddedData[i] := Data[i];
END_FOR;

// Append the bit '1' to the message
PaddedData[Length] := 16#80;

// Append 0 <= k < 512 bits '0', such that the resulting message length in bits
// is congruent to -64 ≡ 448 (mod 512)
PaddedLength := Length + 1;
WHILE (PaddedLength MOD 64) <> 56 DO
    PaddedData[PaddedLength] := 0;
    PaddedLength := PaddedLength + 1;
END_WHILE;

// Append length of message (before pre-processing), in bits, as 64-bit big-endian integer
// Since our message is small (max 127 bytes), we only need the lower 32 bits
Temp := TO_DWORD(Length * 8);
PaddedData[PaddedLength] := 0;
PaddedData[PaddedLength+1] := 0;
PaddedData[PaddedLength+2] := 0;
PaddedData[PaddedLength+3] := 0;
PaddedData[PaddedLength+4] := TO_BYTE(SHR(Temp, 24));
PaddedData[PaddedLength+5] := TO_BYTE(SHR(Temp, 16));
PaddedData[PaddedLength+6] := TO_BYTE(SHR(Temp, 8));
PaddedData[PaddedLength+7] := TO_BYTE(Temp);
PaddedLength := PaddedLength + 8;

NumBlocks := PaddedLength / 64;

// Process the message in successive 512-bit chunks
FOR i := 0 TO NumBlocks - 1 DO
    BlockOffset := i * 64;
    
    // Break chunk into sixteen 32-bit big-endian words w[i], 0 <= i <= 15
    FOR j := 0 TO 15 DO
        W[j] := SHL(TO_DWORD(PaddedData[BlockOffset + j*4]), 24) OR
                SHL(TO_DWORD(PaddedData[BlockOffset + j*4 + 1]), 16) OR
                SHL(TO_DWORD(PaddedData[BlockOffset + j*4 + 2]), 8) OR
                TO_DWORD(PaddedData[BlockOffset + j*4 + 3]);
    END_FOR;
    
    // Message schedule: extend the sixteen 32-bit words into eighty 32-bit words
    FOR j := 16 TO 79 DO
        Temp := W[j-3] XOR W[j-8] XOR W[j-14] XOR W[j-16];
        W[j] := SHL(Temp, 1) OR SHR(Temp, 31); // Left rotate by 1
    END_FOR;
    
    // Initialize hash value for this chunk
    A := H0;
    B := H1;
    C := H2;
    D := H3;
    E := H4;
    
    // Main loop
    FOR j := 0 TO 79 DO
        IF j <= 19 THEN
            F := (B AND C) OR ((NOT B) AND D);
            K := 16#5A827999;
        ELSIF j <= 39 THEN
            F := B XOR C XOR D;
            K := 16#6ED9EBA1;
        ELSIF j <= 59 THEN
            F := (B AND C) OR (B AND D) OR (C AND D);
            K := 16#8F1BBCDC;
        ELSE
            F := B XOR C XOR D;
            K := 16#CA62C1D6;
        END_IF;
        
        Temp := (SHL(A, 5) OR SHR(A, 27)) + F + E + K + W[j];
        E := D;
        D := C;
        C := SHL(B, 30) OR SHR(B, 2);
        B := A;
        A := Temp;
    END_FOR;
    
    // Add this chunk's hash to result so far
    H0 := H0 + A;
    H1 := H1 + B;
    H2 := H2 + C;
    H3 := H3 + D;
    H4 := H4 + E;
END_FOR;

// Produce the final hash value (big-endian)
Hash[0] := TO_BYTE(SHR(H0, 24)); Hash[1] := TO_BYTE(SHR(H0, 16)); Hash[2] := TO_BYTE(SHR(H0, 8)); Hash[3] := TO_BYTE(H0);
Hash[4] := TO_BYTE(SHR(H1, 24)); Hash[5] := TO_BYTE(SHR(H1, 16)); Hash[6] := TO_BYTE(SHR(H1, 8)); Hash[7] := TO_BYTE(H1);
Hash[8] := TO_BYTE(SHR(H2, 24)); Hash[9] := TO_BYTE(SHR(H2, 16)); Hash[10] := TO_BYTE(SHR(H2, 8)); Hash[11] := TO_BYTE(H2);
Hash[12] := TO_BYTE(SHR(H3, 24)); Hash[13] := TO_BYTE(SHR(H3, 16)); Hash[14] := TO_BYTE(SHR(H3, 8)); Hash[15] := TO_BYTE(H3);
Hash[16] := TO_BYTE(SHR(H4, 24)); Hash[17] := TO_BYTE(SHR(H4, 16)); Hash[18] := TO_BYTE(SHR(H4, 8)); Hash[19] := TO_BYTE(H4);
          
END_FUNCTION_BLOCK

FUNCTION_BLOCK FB_CRC32_Calculator
  VAR
    L_Table : ARRAY[0..255] OF DWORD;
    L_Initialized : BOOL := FALSE;
  END_VAR

            METHOD Calculate : DWORD

Calculate := 0;
END_METHOD
          
END_FUNCTION_BLOCK

FUNCTION_BLOCK FB_Heating_Policy_Observer
  VAR_INPUT
    VI_Zone_Occupied : ARRAY[1..GVL_CONSTANTS.C_MAX_ZONES] OF BOOL;
    VI_Zone_Last_Motion_TS : ARRAY[1..GVL_CONSTANTS.C_MAX_ZONES] OF UDINT;
    VI_System_Time_MS : UDINT;
    VI_Zone_Permanent_Use : ARRAY[1..GVL_CONSTANTS.C_MAX_ZONES] OF BOOL;
    VI_Zone_Guest_Preheat : ARRAY[1..GVL_CONSTANTS.C_MAX_ZONES] OF BOOL;
    VI_Behavior_Mode : E_Behavior_Mode;
  END_VAR
  VAR_OUTPUT
    VO_Zone_Empty_Duration_MS : ARRAY[1..GVL_CONSTANTS.C_MAX_ZONES] OF UDINT;
    VO_Zone_Policy_Class : ARRAY[1..GVL_CONSTANTS.C_MAX_ZONES] OF INT;
    VO_Zone_Target_Adjustment : ARRAY[1..GVL_CONSTANTS.C_MAX_ZONES] OF REAL;
    VO_Zone_Priority_Bias : ARRAY[1..GVL_CONSTANTS.C_MAX_ZONES] OF REAL;
  END_VAR
  VAR
    L_i : INT;
    L_Long_Threshold : UDINT := 86400000;
    L_Away_Mode : BOOL;
  END_VAR

            L_Away_Mode := (VI_Behavior_Mode = BEHAVIOR_AWAY);

FOR L_i := 1 TO GVL_CONSTANTS.C_MAX_ZONES DO

    // compute empty duration
    IF VI_Zone_Occupied[L_i] THEN
        VO_Zone_Empty_Duration_MS[L_i] := 0;
    ELSE
        VO_Zone_Empty_Duration_MS[L_i] := VI_System_Time_MS - VI_Zone_Last_Motion_TS[L_i];
    END_IF;

    // policy classification
    // Guest/preheat has priority even in AWAY mode.
    IF VI_Zone_Guest_Preheat[L_i] THEN
        VO_Zone_Policy_Class[L_i] := 3; // guest

    ELSIF VI_Zone_Occupied[L_i] THEN
        VO_Zone_Policy_Class[L_i] := 0; // comfort

    ELSIF VI_Zone_Permanent_Use[L_i] AND (NOT L_Away_Mode) THEN
        VO_Zone_Policy_Class[L_i] := 4; // permanent mild eco

    ELSIF VO_Zone_Empty_Duration_MS[L_i] >= L_Long_Threshold THEN
        VO_Zone_Policy_Class[L_i] := 2; // deep eco

    ELSE
        VO_Zone_Policy_Class[L_i] := 1; // mild eco
    END_IF;

